(* IEC 61131-3 sources: Trae_CLoudTest/_archive/2026-04-25_全局规范修订V4.1.0/旧版程序文件, 5 files *)

(* ---- FB_单层输送机_V4.0.1.st ---- *)
//==============================================================================
// 边框缓存机 PLC程序 - 单层输送机纯逻辑功能块
// 版本: V4.0.1 (修正计时器使用方式 - 严格按三菱GX Works3标准)
// 项目: DJ-2026-005 边框缓存机
// 编制日期: 2026-04-23
// 更新日期: 2026-04-25 (修正计时器使用规范)
// 遵循规范: IEC 61131-3, 810_PLC编程规范_DEV-V1.0.0, 三菱GX Works3标准
//
// 说明:
//   纯逻辑功能块 - 单层输送机独立控制(不包含任何X/Y/M/D地址引用)
//   所有输入来自主控(已映射的逻辑变量), 所有输出给主控(由主控映射到Y地址)
//
// 功能:
//   1. 9步自动模式状态机控制
//   2. 手动模式点动控制(6个手动操作)
//   3. 初始化流程(气缸复位、状态清零)
//   4. 块内报警检测与处理(7种报警类型)
//   5. 完全自包含,无外部物理地址依赖,无ARRAY,纯单层设计
//
// 架构特点:
//   - 纯逻辑块: 不包含任何X/Y/M/D地址引用
//   - 数据解耦: 通过逻辑变量接口与主控交互
//   - 单层设计: 无ARRAY,所有信号均为单个BOOL/INT/REAL
//   - 故障安全: 内置超时保护和传感器冲突检测
//   - 下游联动: 支持上游允许放料信号和下游放料完成信号交互
//
// ⭐ 计时器使用规范 (V4.0.1 - 严格模仿三菱TIMER_100_FB_M_1):
//   参考原始程序:
//     TIMER_100_FB_M_1(MM[0] & NOT 异常暂停信号, 100, 0, TT1[0], MM[1]);
//     TIMER_100_FB_M_2(MM[2] & NOT 异常暂停信号, TT0[7], 0, TT1[1], MM[3]);
//
//   标准用法:
//     1. 程序开头统一调用TON实例(类似TIMER_100_FB_M_x调用)
//     2. 使用中间BOOL变量控制启动/停止(类似MM[x]:=1/0)
//     3. 使用中间BOOL变量判断到时(类似IF MM[y])
//     4. CASE状态机逻辑中只读写这些中间变量,不直接调用TON
//==============================================================================

FUNCTION_BLOCK FB_单层输送机_V4.0.1

VAR_INPUT
    (*==========================================================================
      一、系统控制信号 (来自主控/HMI M区) - 遵循801规范: i_前缀
      ==========================================================================*)
    i_bEnable            : BOOL;    // 总使能信号(主控系统就绪后置位)

    (*-------------------------------------------------------------------------
      模式选择 (互斥信号,来自HMI M区)
      -------------------------------------------------------------------------*)
    i_bAutoMode          : BOOL;    // 自动运行模式选择
    i_bManualMode        : BOOL;    // 手动调试模式选择

    (*-------------------------------------------------------------------------
      操作按钮 (来自HMI,边沿触发)
      -------------------------------------------------------------------------*)
    i_bStart             : BOOL;    // 自动循环启动按钮
    i_bStop              : BOOL;    // 自动循环停止按钮
    i_bReset             : BOOL;    // 故障复位/初始化按钮

    (*==========================================================================
      二、手动操作信号 (6个BOOL,来自HMI) - 遵循801规范: i_bLx_前缀(HMI辅助)
      ==========================================================================*)
    i_bLx_BlockDown      : BOOL;    // 手动-阻挡气缸下降
    i_bLx_BlockUp        : BOOL;    // 手动-阻挡气缸上升
    i_bLx_SeparatePush   : BOOL;    // 手动-分料气缸推出
    i_bLx_SeparateReset  : BOOL;    // 手动-分料气缸复位
    i_bLx_ConveyorFwd    : BOOL;    // 手动-输送带正转
    i_bLx_ConveyorRev    : BOOL;    // 手动-输送带反转

    (*==========================================================================
      三、工艺参数 (来自HMI设定或配方)
      ==========================================================================*)
    i_rConveyorSpeed     : REAL;    // 输送带速度设定(Hz或m/min,给变频器用)
    i_iSeparateTime      : INT;     // 分料动作保持时间(ms)
    i_iBlockWaitTime     : INT;     // 阻挡气缸动作等待时间(ms)

    (*==========================================================================
      四、传感器输入 (7个BOOL,全部来自主控映射)
      注: 放料完成感应器通过下游信号o_bFeedComplete反馈
      ==========================================================================*)
    (*--- 分料前感应器: 检测材料是否到达分料工位入口 ---*)
    i_bPreSeparateSensor : BOOL;

    (*--- 到位感应器1/2: 双传感器冗余检测材料到位 ---*)
    i_bPositionSensor1   : BOOL;
    i_bPositionSensor2   : BOOL;

    (*--- 阻挡气缸位置反馈 ---*)
    i_bBlockCylinderUp   : BOOL;    // 阻挡升起(释放)位置
    i_bBlockCylinderDown : BOOL;    // 阻挡下降(阻挡)位置

    (*--- 分料气缸位置反馈 ---*)
    i_bSeparateCylinderUp   : BOOL; // 分料收回位置
    i_bSeparateCylinderDown : BOOL; // 分料推出位置

    (*==========================================================================
      五、上下游联锁信号
      ==========================================================================*)
    i_bUpstreamAllowFeed : BOOL;    // 取放料机构已取走,允许继续放料
END_VAR

VAR_OUTPUT
    (*==========================================================================
      一、执行器请求输出 (5个BOOL,全部给主控,由主控映射到Y地址)
      ==========================================================================*)
    o_bBlockSolenoid     : BOOL;    // TRUE=下降(阻挡), FALSE=上升(释放)
    o_bSeparateSolenoid  : BOOL;    // TRUE=推出(分料), FALSE=复位
    o_bConveyorFwd       : BOOL;    // 输送带正向运转
    o_bConveyorSlow      : BOOL;    // 输送带慢速运转(精确定位用)
    o_bConveyorRev       : BOOL;    // 输送带反向运转(退料用)

    (*==========================================================================
      二、下游信号输出 (给取放料机构/打胶机)
      ==========================================================================*)
    o_bFeedComplete      : BOOL;    // 该层放料完成,可取料

    (*==========================================================================
      三、状态/HMI显示输出
      ==========================================================================*)
    o_bRunning           : BOOL;    // 正在自动运行
    o_bFault             : BOOL;    // 本站有故障(报警激活)
    o_iCurrentState      : INT;     // 当前状态码(0=空闲,1-8=步序,99=故障)

    (*==========================================================================
      四、报警输出 (给公共报警管理器)
      ==========================================================================*)
    o_iAlarmCode         : INT;     // 当前有效报警代码(0=无报警,1-7=报警类型)
                                    // 1=阻挡下降超时,2=上升超时,
                                    // 3=分料推出超时,4=复位超时,
                                    // 5=输送超时,6=传感器冲突,7=变频器故障
END_VAR

(*==============================================================================
 内部变量定义 - 遵循801规范: 不加前缀,直接 类型_描述
 ==============================================================================*)
VAR
    (*--------------------------------------------------------------------------
      一、状态机变量
      --------------------------------------------------------------------------*)
    iStep                : INT;     // 当前步序 (0-8)

    (*--- 运行标志 ---*)
    bRunning             : BOOL;    // 正在自动运行标志
    bFault               : BOOL;    // 故障标志

    (*--- 启动触发锁存 (防止重复触发) ---*)
    bStartTriggered       : BOOL;    // 启动信号锁存

    (*--------------------------------------------------------------------------
      二、⭐ 计时器相关变量 - 按三菱标准+801规范命名

      三菱标准接口:
        i_bTime  : BOOL  - 定时器启动输入 (Coil, 类似MM[x])
        q_bTq    : BOOL  - 定时器到时输出 (Status, 类似MM[y])
        i_bTrst  : BOOL  - 定时器复位信号
        i_pTimer : DINT - 定时器预设值 (Preset, 类似TT0[z])
        q_eTimer : DINT - 定时器当前值 (ValueOut, 类似TT1[w])

      801规范前缀:
        i_ = 输入变量 (VAR_INPUT风格,用于内部接口)
        q_ = 输出变量 (VAR_OUTPUT风格,用于内部接口)
      --------------------------------------------------------------------------*)

    (*--- TON计时器实例 (在VAR区声明,类似程序开头的TIMER_100_FB_M_x调用) ---*)
    tTimerAction         : TON;     // 动作等待定时器(阻挡/分料)
    tTimerConveyor       : TON;     // 输送超时定时器
    tTimerReset          : TON;     // 复位等待定时器
    tTimerPulse          : TON;     // 放料完成脉冲定时器(500ms)
    tTimerInit           : TON;     // 初始化总超时定时器

    (*--- 计时器接口变量 (严格按三菱标准命名) ---*)

    (* 启动输入: 写入TRUE=启动, 写入FALSE=停止 (类似 MM[x]:=1/0) *)
    i_bTime_Action       : BOOL;    // 动作定时器启动
    i_bTime_Conveyor     : BOOL;    // 输送定时器启动
    i_bTime_Reset        : BOOL;    // 复位定时器启动
    i_bTime_Pulse        : BOOL;    // 脉冲定时器启动
    i_bTime_Init         : BOOL;    // 初始化定时器启动

    (* 到时输出: 读取判断是否到时 (类似 IF MM[y]) *)
    q_bTq_Action         : BOOL;    // 动作定时器到时
    q_bTq_Conveyor       : BOOL;    // 输送定时器到时
    q_bTq_Reset          : BOOL;    // 复位定时器到时
    q_bTq_Pulse          : BOOL;    // 脉冲定时器到时
    q_bTq_Init           : BOOL;    // 初始化定时器到时

    (* 复位信号: 强制清零当前值 *)
    i_bTrst_Action       : BOOL;    // 动作定时器复位
    i_bTrst_Conveyor     : BOOL;    // 输送定时器复位

    (* 预设值: 可选,用于调试显示 (类似读取TT0[z]) *)
    i_pTimer_Action      : INT;     // 动作定时器预设值(ms)
    i_pTimer_Conveyor    : INT;     // 输送定时器预设值(ms)

    (* 当前值: 可选,用于调试显示 (类似读取TT1[w]) *)
    q_eTimer_Action      : INT;     // 动作定时器当前值(ms)
    q_eTimer_Conveyor    : INT;     // 输送定时器当前值(ms)

    (*--------------------------------------------------------------------------
      三、系统级内部变量
      --------------------------------------------------------------------------*)
    bInitComplete        : BOOL;    // 上电初始化完成标志
    bInitInProgress      : BOOL;    // 正在执行初始化

    (*--- 报警相关 ---*)
    iActiveAlarm         : INT;     // 当前活跃报警代码

    (*--- 传感器冲突检测 ---*)
    bBlockConflict       : BOOL;    // 阻挡上下位同时为TRUE
    bSeparateConflict    : BOOL;    // 分料上下位同时为TRUE

    (*--- 手动操作互锁 ---*)
    bManualAllow         : BOOL;    // 允许手动操作标志
END_VAR

(*==============================================================================
 常量定义 (状态机步序 + 报警码 + 定时参数)
 ==============================================================================*)
VAR CONSTANT
    (*--------------------------------------------------------------------------
      状态机步序常量 (9步: 0空闲 + 8工作步)
      --------------------------------------------------------------------------*)
    STP_IDLE             : INT := 0;   // 空闲待机
    STP_DETECT_MATERIAL  : INT := 1;   // 等待分料前感应器信号
    STP_BLOCK_DOWN       : INT := 2;   // 阻挡气缸下降到位
    STP_CONVEYOR_FWD     : INT := 3;   // 输送带正转运料
    STP_POSITION_CHECK   : INT := 4;   // 等待双传感器到位确认
    STP_BLOCK_UP         : INT := 5;   // 阻挡气缸上升释放
    STP_SEPARATE_ACTION  : INT := 6;   // 分料气缸推出分离
    STP_SLOW_FEED        : INT := 7;   // 慢速精确送出
    STP_FEED_COMPLETE    : INT := 8;   // 放料完成,等待取料

    (*--------------------------------------------------------------------------
      报警码常量 (1~7段,0=无报警)
      --------------------------------------------------------------------------*)
    ALM_BLOCK_DOWN_TIMEOUT   : INT := 1;
    ALM_BLOCK_UP_TIMEOUT    : INT := 2;
    ALM_SEPARATE_PUSH_TIMEOUT : INT := 3;
    ALM_SEPARATE_RESET_TIMEOUT : INT := 4;
    ALM_CONVEYOR_TIMEOUT    : INT := 5;
    ALM_SENSOR_CONFLICT     : INT := 6;
    ALM_INVERTER_FAULT      : INT := 7;

    (*--------------------------------------------------------------------------
      默认定时参数 (单位: ms,可通过输入参数覆盖)
      --------------------------------------------------------------------------*)
    T_DEF_BLOCK_ACTION_TIME     : INT := 800;    // 阻挡气缸动作时间
    T_DEF_SEPARATE_ACTION_TIME  : INT := 1000;   // 分料气缸动作时间
    T_DEF_CONVEYOR_TIMEOUT_TIME : INT := 5000;   // 输送带超时保护
    T_DEF_POSITION_STABLE_TIME  : INT := 500;    // 到位后稳定等待
    T_DEF_SLOW_FEED_TIME        : INT := 2000;   // 慢速送出时间
    T_DEF_RESET_WAIT_TIME       : INT := 500;    // 复位等待时间
    T_DEF_INIT_TIMEOUT          : INT := 10000;  // 初始化总超时(10s)
    T_DEF_FEED_PULSE_TIME       : INT := 500;    // 放料完成脉冲宽度(ms)
END_VAR

(*==============================================================================
 主程序开始 - 执行顺序说明 (严格模仿三菱原始程序结构):

   第一部分: 使能与初始化处理
   第二部分: 传感器冲突检测
   第三部分: 模式分发 (自动/手动)
   第四部分: 停止与复位处理
   第五部分: ⭐ TON统一实例化 (模仿TIMER_100_FB_M_x调用)
   第六部分: 状态机逻辑 (只操作bTimerXXX_Done接口,不直接调用TON)
   第七部分: 状态输出汇总
 ==============================================================================*)

//==============================================================================
// 第一部分: 使能与初始化处理
//==============================================================================

(*--- 使能失效时的安全处理 ---*)
IF NOT i_bEnable THEN
    (* 清零所有输出 *)
    o_bBlockSolenoid    := FALSE;
    o_bSeparateSolenoid := FALSE;
    o_bConveyorFwd      := FALSE;
    o_bConveyorSlow     := FALSE;
    o_bConveyorRev      := FALSE;
    o_bFeedComplete     := FALSE;

    (* 清零状态 *)
    iStep               := STP_IDLE;
    bRunning            := FALSE;
    bFault              := FALSE;
    bStartTriggered     := FALSE;
    iActiveAlarm        := 0;
    bInitComplete       := FALSE;
    bInitInProgress     := FALSE;

    (* 清零输出状态 *)
    o_bRunning          := FALSE;
    o_bFault            := FALSE;
    o_iCurrentState     := STP_IDLE;
    o_iAlarmCode        := 0;

    (* ⭐ 停止所有计时器 (清除启动标志,类似 MM[x]:=0) *)
    i_bTime_Action   := FALSE;
    i_bTime_Conveyor := FALSE;
    i_bTime_Reset    := FALSE;
    i_bTime_Pulse    := FALSE;
    i_bTime_Init     := FALSE;

    RETURN;  (* 退出功能块,不执行后续逻辑 *)
END_IF;

//==============================================================================
// 第二部分: 初始化流程 (上电或复位后首次使能时执行)
//==============================================================================

IF NOT bInitComplete THEN
    bInitInProgress := TRUE;

    (* ⭐ 启动初始化计时器 (设置启动标志,类似 MM[x]:=1) *)
    i_bTime_Init := TRUE;

    (* 执行初始化: 气缸回到安全位置 *)
    (* 阻挡电磁阀OFF -> 阻挡上升到上位 *)
    o_bBlockSolenoid    := FALSE;
    (* 分料电磁阀OFF -> 分料气缸复位到上位 *)
    o_bSeparateSolenoid := FALSE;
    (* 输送带全部停止 *)
    o_bConveyorFwd      := FALSE;
    o_bConveyorSlow     := FALSE;
    o_bConveyorRev      := FALSE;
    (* 步序归零 *)
    iStep               := STP_IDLE;
    bFault              := FALSE;
    iActiveAlarm        := 0;

    (* 检查初始化条件: 阻挡在上位 AND 分料在上位 OR 超时强制完成 *)
    IF (i_bBlockCylinderUp AND i_bSeparateCylinderUp) OR q_bTq_Init THEN
        (* 初始化完成 或 超时强制完成 *)
        bInitComplete   := TRUE;
        bInitInProgress := FALSE;
        (* ⭐ 停止初始化计时器 (清除启动标志,类似 MM[x]:=0) *)
        i_bTime_Init := FALSE;
    END_IF;

    (* 初始化期间不执行自动/手动逻辑 *)
    o_bRunning      := FALSE;
    o_iCurrentState := STP_IDLE;
    RETURN;
END_IF;

//==============================================================================
// 第三部分: 传感器冲突检测 (所有模式共用)
//==============================================================================

(* 阻挡气缸上下位同时为TRUE -> 传感器故障或接线错误 *)
bBlockConflict := i_bBlockCylinderUp AND i_bBlockCylinderDown;

(* 分料气缸上下位同时为TRUE -> 传感器故障或接线错误 *)
bSeparateConflict := i_bSeparateCylinderUp AND i_bSeparateCylinderDown;

(* 记录传感器冲突报警 *)
IF bBlockConflict OR bSeparateConflict THEN
    iActiveAlarm := ALM_SENSOR_CONFLICT;
    bFault      := TRUE;
ELSIF iActiveAlarm = ALM_SENSOR_CONFLICT THEN
    (* 冲突消失且当前只有此报警 -> 清除 *)
    iActiveAlarm := 0;
    bFault      := FALSE;
END_IF;

//==============================================================================
// 第四部分: 模式分发 (自动/手动)
//==============================================================================

IF i_bAutoMode THEN
    (*==========================================================================
      自动模式: 执行9步状态机
      =========================================================================*)
    CALL_AutoModeStateMachine();

ELSIF i_bManualMode THEN
    (*==========================================================================
      手动模式: 执行手动点动控制
      =========================================================================*)
    CALL_ManualModeControl();

ELSE
    (* 无效模式: 停止所有输出 *)
    o_bBlockSolenoid    := FALSE;
    o_bSeparateSolenoid := FALSE;
    o_bConveyorFwd      := FALSE;
    o_bConveyorSlow     := FALSE;
    o_bConveyorRev      := FALSE;
    o_bFeedComplete     := FALSE;

    (* 如果不在故障态,归零步序 *)
    IF NOT bFault THEN
        iStep := STP_IDLE;
    END_IF;
    bRunning := FALSE;

    (* ⭐ 无效模式下也停止所有计时器 *)
    i_bTime_Action   := FALSE;
    i_bTime_Conveyor := FALSE;
    i_bTime_Reset    := FALSE;
    i_bTime_Pulse    := FALSE;
END_IF;

//==============================================================================
// 第五部分: 停止与复位处理
//==============================================================================

(*--- 全局停止: 停止自动循环 ---*)
IF i_bStop THEN
    IF bRunning AND NOT bFault THEN
        iStep           := STP_IDLE;
        bRunning        := FALSE;
        bStartTriggered := FALSE;

        (* 停止该层输出 *)
        o_bBlockSolenoid    := FALSE;
        o_bSeparateSolenoid := FALSE;
        o_bConveyorFwd      := FALSE;
        o_bConveyorSlow     := FALSE;
        o_bConveyorRev      := FALSE;

        (* ⭐ 停止所有计时器 *)
        i_bTime_Action   := FALSE;
        i_bTime_Conveyor := FALSE;
        i_bTime_Reset    := FALSE;
        i_bTime_Pulse    := FALSE;
    END_IF;
END_IF;

(*--- 全局复位: 清除所有报警和故障 ---*)
IF i_bReset THEN
    IF bFault THEN
        (* 清除报警和故障标志 *)
        iActiveAlarm := 0;
        bFault      := FALSE;

        (* 归零步序 *)
        iStep           := STP_IDLE;
        bRunning        := FALSE;
        bStartTriggered := FALSE;

        (* 安全输出状态 *)
        o_bBlockSolenoid    := FALSE;
        o_bSeparateSolenoid := FALSE;
        o_bConveyorFwd      := FALSE;
        o_bConveyorSlow     := FALSE;
        o_bConveyorRev      := FALSE;
        o_bFeedComplete     := FALSE;

        (* ⭐ 停止所有计时器 *)
        i_bTime_Action   := FALSE;
        i_bTime_Conveyor := FALSE;
        i_bTime_Reset    := FALSE;
        i_bTime_Pulse    := FALSE;

        (* 要求重新初始化 *)
        bInitComplete := FALSE;
    END_IF;
END_IF;

//==============================================================================
// 第五部分: ⭐ TON统一实例化 (严格模仿三菱TIMER_100_FB_M_x模式)
//
// 原始程序格式:
//   TIMER_100_FB_M_1(MM[0] & NOT 异常暂停信号, 100, 0, TT1[0], MM[1]);
//   参数: s1(Coil)=执行条件, s2(Preset)=设定值, s3(ValueIn)=初始值,
//         d1(ValueOut)=当前值, d2(Status)=到时输出
//
// 本实现使用IEC标准TON,但保持相同的使用模式:
//   - 此处统一调用所有TON实例(类似程序开头的5行TIMER调用)
//   - 使用i_bTime_xxx控制IN(类似MM[x])
//   - 将.Q映射到q_bTq_xxx(类似MM[y])
//   - 将.ET映射到q_eTimer_xxx(类似TT1[w])
//==============================================================================

(*--- TON_1: 动作定时器 (阻挡/分料动作等待) ---*)
tTimerAction(
    IN  := i_bTime_Action,
    PT  := T#MS * (
            IF iStep = STP_BLOCK_DOWN AND i_iBlockWaitTime > 0
                THEN i_iBlockWaitTime
            ELSIF iStep = STP_SEPARATE_ACTION AND i_iSeparateTime > 0
                THEN i_iSeparateTime
            ELSIF iStep = STP_POSITION_CHECK
                THEN T_DEF_POSITION_STABLE_TIME
            ELSE
                T_DEF_BLOCK_ACTION_TIME
            END
        )
);

(*--- TON_2: 输送定时器 (输送超时保护) ---*)
tTimerConveyor(
    IN  := i_bTime_Conveyor,
    PT  := T#MS * (
            IF iStep = STP_SLOW_FEED
                THEN T_DEF_SLOW_FEED_TIME
            ELSE
                T_DEF_CONVEYOR_TIMEOUT_TIME
            END
        )
);

(*--- TON_3: 复位定时器 (暂未使用,预留) ---*)
tTimerReset(
    IN  := i_bTime_Reset,
    PT  := T#MS * T_DEF_RESET_WAIT_TIME
);

(*--- TON_4: 放料完成脉冲定时器 (500ms脉冲) ---*)
tTimerPulse(
    IN  := i_bTime_Pulse,
    PT  := T#MS * T_DEF_FEED_PULSE_TIME
);

(*--- TON_5: 初始化定时器 (10s总超时) ---*)
tTimerInit(
    IN  := i_bTime_Init,
    PT  := T#MS * T_DEF_INIT_TIMEOUT
);

(*--- 映射输出接口 (将TON的.Q/.ET映射到标准接口变量) ---*)

(* 到时输出: .Q -> q_bTq_xxx (类似 Status->MM[y]) *)
q_bTq_Action     := tTimerAction.Q;
q_bTq_Conveyor   := tTimerConveyor.Q;
q_bTq_Reset      := tTimerReset.Q;
q_bTq_Pulse      := tTimerPulse.Q;
q_bTq_Init       := tTimerInit.Q;

(* 当前值: .ET -> q_eTimer_xxx (类似 ValueOut->TT1[w]) *)
q_eTimer_Action   := UINT_TO_INT(TIME_TO_UINT(tTimerAction.ET)) / 10;   // 转换为ms
q_eTimer_Conveyor := UINT_TO_INT(TIME_TO_UINT(tTimerConveyor.ET)) / 10;

(* 预设值记录: PT -> i_pTimer_xxx (用于调试显示) *)
i_pTimer_Action   := UINT_TO_INT(TIME_TO_UINT(tTimerAction.PT)) / 10;
i_pTimer_Conveyor := UINT_TO_INT(TIME_TO_UINT(tTimerConveyor.PT)) / 10;

//==============================================================================
// 第六部分: 状态机逻辑 (只操作q_bTq_xxx接口,不直接调用TON)
// 类似原始程序的CASE Step_S OF ... END_CASE部分
//==============================================================================

(*--- 9步状态机主体 (仅使用q_bTq_xxx判断到时,类似IF MM[y]) ---*)
CASE iStep OF

(*======================================================================
 步骤0: 空闲待机
 条件: 启动触发 + 分料前有材料 + 上游允许放料
 ======================================================================*)
STP_IDLE:
    bRunning := FALSE;

    (* 安全输出状态 *)
    o_bBlockSolenoid    := FALSE;
    o_bSeparateSolenoid := FALSE;
    o_bConveyorFwd      := FALSE;
    o_bConveyorSlow     := FALSE;
    o_bConveyorRev      := FALSE;
    o_bFeedComplete     := FALSE;

    (* ⭐ 停止所有计时器 (设置启动标志=FALSE,类似 MM[x]:=0) *)
    i_bTime_Action   := FALSE;
    i_bTime_Conveyor := FALSE;
    i_bTime_Pulse    := FALSE;

    (* 启动条件:
       - 收到启动触发
       - 分料前有材料到位
       - 上游允许放料(取放料机构已取走上一次的材料)
    *)
    IF bStartTriggered AND i_bPreSeparateSensor AND i_bUpstreamAllowFeed THEN
        iStep    := STP_DETECT_MATERIAL;
        bRunning := TRUE;
        (* ⭐ 启动输送计时器 (设置启动标志=TRUE,类似 MM[x]:=1) *)
        i_bTime_Conveyor := TRUE;
    END_IF;

(*======================================================================
 步骤1: 检测材料到位 (双重确认)
 转出条件: 分料前感应器稳定信号
 超时条件: 材料未到达 -> ALM_CONVEYOR_TIMEOUT (检查q_bTq_Conveyor)
 ======================================================================*)
STP_DETECT_MATERIAL:
    (* 等待分料前感应器稳定信号 *)
    IF i_bPreSeparateSensor THEN
        (* 材料确认到位,进入阻挡下降 *)
        iStep := STP_BLOCK_DOWN;
        (* ⭐ 切换到动作计时器 (先停旧的,再启新的) *)
        i_bTime_Conveyor := FALSE;  // 停止输送计时器
        i_bTime_Action := TRUE;     // 启动动作计时器
    ELSIF q_bTq_Conveyor THEN  (* ✅ 读取到时标志,类似 IF MM[3] *)
        (* 超时: 材料未到达 *)
        iActiveAlarm := ALM_CONVEYOR_TIMEOUT;
        bFault       := TRUE;
        iStep        := STP_IDLE;
        bRunning     := FALSE;
        i_bTime_Conveyor := FALSE;  // 停止计时器
    END_IF;

(*======================================================================
 步骤2: 阻挡下降 (等待气缸下位信号或超时)
 动作: 保持o_bBlockSolenoid=TRUE
 转出条件: i_bBlockCylinderDown
 超时条件: ALM_BLOCK_DOWN_TIMEOUT (检查q_bTq_Action)
 ======================================================================*)
STP_BLOCK_DOWN:
    o_bBlockSolenoid := TRUE;  (* 保持下降 *)

    IF i_bBlockCylinderDown THEN
        (* 阻挡到位,转入输送 *)
        iStep := STP_CONVEYOR_FWD;
        o_bConveyorFwd := TRUE;
        (* ⭐ 切换到输送计时器 *)
        i_bTime_Action := FALSE;
        i_bTime_Conveyor := TRUE;
    ELSIF q_bTq_Action THEN  (* ✅ 读取到时标志,类似 IF MM[1] *)
        (* 超时: 阻挡未到位 *)
        iActiveAlarm := ALM_BLOCK_DOWN_TIMEOUT;
        bFault       := TRUE;
        o_bBlockSolenoid := FALSE;
        iStep        := STP_IDLE;
        bRunning     := FALSE;
        i_bTime_Action := FALSE;
    END_IF;

(*======================================================================
 步骤3: 输送正转 (将材料送到到位传感器位置)
 动作: 保持o_bConveyorFwd=TRUE
 转出条件: i_bPositionSensor1 AND i_bPositionSensor2 (双传感器冗余)
 超时条件: ALM_CONVEYOR_TIMEOUT (检查q_bTq_Conveyor)
 ======================================================================*)
STP_CONVEYOR_FWD:
    o_bConveyorFwd := TRUE;  (* 保持正转 *)

    (* 双传感器都到位 -> 输送成功 *)
    IF i_bPositionSensor1 AND i_bPositionSensor2 THEN
        iStep := STP_POSITION_CHECK;
        o_bConveyorFwd := FALSE;  (* 停止输送 *)
        (* ⭐ 切换到动作计时器(到位稳定等待) *)
        i_bTime_Conveyor := FALSE;
        i_bTime_Action := TRUE;
    ELSIF q_bTq_Conveyor THEN  (* ✅ 读取到时标志 *)
        (* 超时: 输送未到位 *)
        iActiveAlarm := ALM_CONVEYOR_TIMEOUT;
        bFault       := TRUE;
        o_bConveyorFwd := FALSE;
        iStep        := STP_IDLE;
        bRunning     := FALSE;
        i_bTime_Conveyor := FALSE;
    END_IF;

(*======================================================================
 步骤4: 到位检测 (短暂稳定等待后进入阻挡上升)
 动作: 保持阻挡,全部输出关闭,等待稳定
 转出条件: 定时器到期 (检查q_bTq_Action)
 ======================================================================*)
STP_POSITION_CHECK:
    (* 全部输出保持关闭,等待稳定,但保持阻挡 *)
    o_bBlockSolenoid := TRUE;  (* 保持阻挡 *)

    IF q_bTq_Action THEN  (* ✅ 读取到时标志 *)
        iStep := STP_BLOCK_UP;
        (* 开始阻挡上升(释放) *)
        o_bBlockSolenoid := FALSE;  (* OFF=上升 *)
        (* ⭐ 继续使用动作计时器(阻挡上升等待) - PT会自动根据iStep调整 *)
    END_IF;

(*======================================================================
 步骤5: 阻挡上升 (释放材料,准备分料)
 动作: 保持o_bBlockSolenoid=FALSE (上升状态)
 转出条件: i_bBlockCylinderUp
 超时条件: ALM_BLOCK_UP_TIMEOUT (检查q_bTq_Action)
 ======================================================================*)
STP_BLOCK_UP:
    o_bBlockSolenoid := FALSE;  (* 保持上升状态 *)

    IF i_bBlockCylinderUp THEN
        (* 阻挡已上升,进入分料 *)
        iStep := STP_SEPARATE_ACTION;
        o_bSeparateSolenoid := TRUE;  (* 推出分料 *)
        (* ⭐ 继续使用动作计时器(分料动作等待) *)
    ELSIF q_bTq_Action THEN  (* ✅ 读取到时标志 *)
        (* 超时: 阻挡未上升 *)
        iActiveAlarm := ALM_BLOCK_UP_TIMEOUT;
        bFault       := TRUE;
        iStep        := STP_IDLE;
        bRunning     := FALSE;
        i_bTime_Action := FALSE;
    END_IF;

(*======================================================================
 步骤6: 分料动作 (分料气缸推出,将材料分离)
 动作: 保持o_bSeparateSolenoid=TRUE
 转出条件: i_bSeparateCylinderDown
 超时条件: ALM_SEPARATE_PUSH_TIMEOUT (检查q_bTq_Action)
 ======================================================================*)
STP_SEPARATE_ACTION:
    o_bSeparateSolenoid := TRUE;  (* 保持推出 *)

    IF i_bSeparateCylinderDown THEN
        (* 分料到位,转入慢速送出 *)
        iStep := STP_SLOW_FEED;
        o_bSeparateSolenoid := FALSE;  (* 开始复位 *)
        o_bConveyorSlow := TRUE;  (* 慢速送出 *)
        (* ⭐ 切换到输送计时器(慢速送出等待) *)
        i_bTime_Action := FALSE;
        i_bTime_Conveyor := TRUE;
    ELSIF q_bTq_Action THEN  (* ✅ 读取到时标志 *)
        (* 超时: 分料未到位 *)
        iActiveAlarm := ALM_SEPARATE_PUSH_TIMEOUT;
        bFault       := TRUE;
        o_bSeparateSolenoid := FALSE;
        iStep        := STP_IDLE;
        bRunning     := FALSE;
        i_bTime_Action := FALSE;
    END_IF;

(*======================================================================
 步骤7: 慢速送出 (精确送出到取料位置)
 动作: o_bConveyorSlow=TRUE, o_bSeparateSolenoid=FALSE(持续复位)
 转出条件: 定时器到期 + 分料已复位验证 (检查q_bTq_Conveyor)
 超时/异常: ALM_SEPARATE_RESET_TIMEOUT
 ======================================================================*)
STP_SLOW_FEED:
    o_bConveyorSlow     := TRUE;   (* 保持慢速 *)
    o_bSeparateSolenoid := FALSE;  (* 分料持续复位 *)

    (* 检查慢速送出时间到 *)
    IF q_bTq_Conveyor THEN  (* ✅ 读取到时标志 *)

        (* 验证分料气缸是否已复位 *)
        IF NOT i_bSeparateCylinderDown OR i_bSeparateCylinderUp THEN
            (* 正常: 分料已复位或在下位信号消失 *)
            iStep := STP_FEED_COMPLETE;
            o_bConveyorSlow := FALSE;
            o_bFeedComplete := TRUE;  (* 通知下游可取料 *)
            (* ⭐ 切换到脉冲计时器 *)
            i_bTime_Conveyor := FALSE;
            i_bTime_Pulse := TRUE;
        ELSE
            (* 异常: 分料气缸卡在推出位置 *)
            iActiveAlarm := ALM_SEPARATE_RESET_TIMEOUT;
            bFault       := TRUE;
            o_bConveyorSlow := FALSE;
            iStep        := STP_IDLE;
            bRunning     := FALSE;
            i_bTime_Conveyor := FALSE;
        END_IF;
    END_IF;

(*======================================================================
 步骤8: 放料完成 (等待下游取料完成后回到空闲)
 动作: 保持o_bFeedComplete=TRUE (脉冲500ms或直到下游确认)
 转出条件: 启动触发被消耗(下一轮启动可重新开始)
 ======================================================================*)
STP_FEED_COMPLETE:
    (* 放料完成脉冲控制: 保持500ms后自动结束 *)
    IF q_bTq_Pulse THEN  (* ✅ 读取到时标志 *)
        iStep           := STP_IDLE;
        bRunning        := FALSE;
        o_bFeedComplete := FALSE;
        bStartTriggered := FALSE;  (* 消耗启动触发,准备接收下一次 *)
        i_bTime_Pulse := FALSE;  (* 停止脉冲计时器 *)
    ELSE
        o_bFeedComplete := TRUE;  (* 保持放料完成信号 *)
    END_IF;

ELSE
    (* 无效步序: 强制归零 *)
    iStep   := STP_IDLE;
    bRunning := FALSE;
    (* 停止所有计时器 *)
    i_bTime_Action   := FALSE;
    i_bTime_Conveyor := FALSE;
    i_bTime_Reset    := FALSE;
    i_bTime_Pulse    := FALSE;

END_CASE;

//==============================================================================
// 第七部分: 状态输出汇总
//==============================================================================

(*--- 运行中标志 ---*)
o_bRunning := bRunning;

(*--- 故障标志 ---*)
o_bFault := bFault;

(*--- 当前状态: 有故障则返回99,否则返回当前步序 ---*)
IF bFault THEN
    o_iCurrentState := 99;
ELSE
    o_iCurrentState := iStep;
END_IF;

(*--- 报警代码输出 ---*)
o_iAlarmCode := iActiveAlarm;

(*==============================================================================
 子程序: 自动模式状态机 (9步完整流程)
 注意: 实际的状态机逻辑已在第六部分的CASE语句中实现
 此子程序保留用于未来扩展或复杂逻辑封装
 ==============================================================================*)
METHOD CALL_AutoModeStateMachine : VOID
    (* 状态机主体已在主程序第六部分实现,此处无需重复代码 *)
    (* 如需封装,可将第六部分的CASE语句移至此处 *)
END_METHOD

(*==============================================================================
 子程序: 手动模式控制 (6个手动操作,带互锁和安全限制)
  ==============================================================================*)
METHOD CALL_ManualModeControl : VOID

    (* 故障层禁止手动操作 *)
    IF bFault THEN
        bManualAllow      := FALSE;
        o_bBlockSolenoid  := FALSE;
        o_bSeparateSolenoid := FALSE;
        o_bConveyorFwd    := FALSE;
        o_bConveyorSlow   := FALSE;
        o_bConveyorRev    := FALSE;
        iStep             := STP_IDLE;

        (* 停止所有计时器 *)
        i_bTime_Action   := FALSE;
        i_bTime_Conveyor := FALSE;
        i_bTime_Reset    := FALSE;
        i_bTime_Pulse    := FALSE;

        RETURN;
    END_IF;

    bManualAllow := TRUE;
    bRunning     := FALSE;
    iStep        := STP_IDLE;  (* 手动模式下步序显示为空闲 *)
    o_bFeedComplete := FALSE;

    (* 停止所有自动计时器 *)
    i_bTime_Action   := FALSE;
    i_bTime_Conveyor := FALSE;
    i_bTime_Pulse    := FALSE;

    (*======================================================================
     手动操作 - 阻挡气缸控制 (互锁: 下降/上升不能同时)
     ======================================================================*)
    IF i_bLx_BlockDown AND NOT i_bLx_BlockUp THEN
        (* 下降请求 *)
        o_bBlockSolenoid := TRUE;  (* 下降 *)
    ELSIF i_bLx_BlockUp AND NOT i_bLx_BlockDown THEN
        (* 上升请求 *)
        o_bBlockSolenoid := FALSE;  (* 上升 *)
    ELSE
        (* 无操作: 保持当前位置 *)
    END_IF;

    (*======================================================================
     手动操作 - 分料气缸控制 (互锁: 推出/复位不能同时)
     ======================================================================*)
    IF i_bLx_SeparatePush AND NOT i_bLx_SeparateReset THEN
        (* 推出请求 *)
        o_bSeparateSolenoid := TRUE;  (* 推出 *)
    ELSIF i_bLx_SeparateReset AND NOT i_bLx_SeparatePush THEN
        (* 复位请求 *)
        o_bSeparateSolenoid := FALSE;  (* 复位 *)
    ELSE
        (* 无操作 *)
    END_IF;

    (*======================================================================
     手动操作 - 输送带控制 (互锁: 正转/反转不能同时,慢速可叠加)
     ======================================================================*)
    IF i_bLx_ConveyorFwd AND NOT i_bLx_ConveyorRev THEN
        o_bConveyorFwd := TRUE;
        o_bConveyorRev := FALSE;
    ELSIF i_bLx_ConveyorRev AND NOT i_bLx_ConveyorFwd THEN
        o_bConveyorFwd := FALSE;
        o_bConveyorRev := TRUE;
    ELSE
        (* 正转/反转都没按: 停止输送 *)
        o_bConveyorFwd := FALSE;
        o_bConveyorRev := FALSE;
    END_IF;

    (* 慢速可作为独立控制或与正转叠加(根据实际工艺需求调整) *)
    (* 此处默认: 手动模式下慢速由外部单独控制或与正转联动 *)
    o_bConveyorSlow := FALSE;  (* 手动模式下默认不用慢速,可按需修改 *)

END_FUNCTION_BLOCK

//==============================================================================
// 程序结束
//==============================================================================

(* ---- FB_取放料机构_V4.0.0.st ---- *)
//==============================================================================
// 边框缓存机 PLC程序 - 取放料机构纯逻辑功能块
// 版本: V4.0.0
// 项目: DJ-2026-005 边框缓存机
// 编制日期: 2026-04-23
// 遵循规范: IEC 61131-3, 810_PLC编程规范_DEV-V1.0.0
// 说明: 纯逻辑功能块 - 取放料机构独立控制(不包含任何X/Y/M/D地址引用)
//       所有输入来自主控(已映射的逻辑变量), 所有输出给主控(由主控映射到Y地址)
//
// 核心工艺:
//   一次取两根边框(前后夹紧同时动作), 4层总共循环取2次
//   取料顺序: 第1次取L1+L2层, 第2次取L3+L4层
//   每次取料后移动到放料位置, 完成放料后通知下游(打胶机送料机构)
//
// 架构特点:
//   - 纯逻辑块: 不包含任何X/Y/M/D地址引用
//   - 数据解耦: 通过逻辑变量接口与主控交互
//   - 11步状态机: 完整的自动取放料循环控制
//   - 故障安全: 内置超时保护、伺服故障检测、传感器冲突检测
//   - 4层循环: 自动管理4层取放料进度, 循环2次完成全部取料
//==============================================================================

//==============================================================================
// 功能块: FB_取放料机构 - 取放料机构纯逻辑控制
// 功能:
//   1. 自动模式状态机(11步完整取放料循环)
//   2. 手动模式控制(14个手动操作信号)
//   3. 初始化流程(气缸复位、伺服使能、状态清零)
//   4. 块内报警检测与处理(8种报警类型, 101~199段)
//   5. 4层循环计数器(一次取两层, 循环2次取完4层)
//   6. 完全自包含, 无外部物理地址依赖
//==============================================================================
FUNCTION_BLOCK FB_1003_PickPlace_BufferFraming

VAR_INPUT
    (*==========================================================================
      一、系统控制信号 (来自主控/HMI M区)
      ==========================================================================*)
    i_b使能               : BOOL;    // 总使能信号(主控系统就绪后置位)

    (*-------------------------------------------------------------------------
      模式选择 (互斥信号,来自HMI M区)
      -------------------------------------------------------------------------*)
    i_b自动模式           : BOOL;    // 自动运行模式选择
    i_b手动模式           : BOOL;    // 手动调试模式选择

    (*-------------------------------------------------------------------------
      操作按钮 (来自HMI,边沿触发或电平有效)
      -------------------------------------------------------------------------*)
    i_b启动               : BOOL;    // 自动循环启动按钮(上升沿触发)
    i_b停止               : BOOL;    // 自动循环停止按钮(电平有效)
    i_b复位               : BOOL;    // 故障复位/初始化按钮(电平有效)

    (*==========================================================================
      二、手动操作信号 (14个BOOL,来自HMI)
      ==========================================================================*)
    (*--- 伺服点动控制 (4个) ---*)
    i_bZ轴点动上          : BOOL;    // 手动-Z轴向上点动
    i_bZ轴点动下          : BOOL;    // 手动-Z轴向下点动
    i_bX1轴点动前         : BOOL;    // 手动-X1轴向前点动(取料方向)
    i_bX1轴点动后         : BOOL;    // 手动-X1轴向后点动(放料方向)

    (*--- 气缸手动控制 (10个) ---*)
    (* 升降气缸: 双电磁阀控制 *)
    i_b升降上升           : BOOL;    // 手动-升降气缸上升
    i_b升降下降           : BOOL;    // 手动-升降气缸下降

    (* 前夹紧气缸: 双电磁阀控制(夹紧/松开) *)
    i_b前夹紧夹紧         : BOOL;    // 手动-前夹紧气缸夹紧
    i_b前夹紧松开         : BOOL;    // 手动-前夹紧气缸松开

    (* 后夹紧气缸: 双电磁阀控制(夹紧/松开) *)
    i_b后夹紧夹紧         : BOOL;    // 手动-后夹紧气缸夹紧
    i_b后夹紧松开         : BOOL;    // 手动-后夹紧气缸松开

    (* 前夹紧2气缸: 双电磁阀控制(夹紧/松开) - 第二组前夹爪 *)
    i_b前夹紧2夹紧        : BOOL;    // 手动-前夹紧2气缸夹紧
    i_b前夹紧2松开        : BOOL;    // 手动-前夹紧2气缸松开

    (* 后夹紧2气缸: 双电磁阀控制(夹紧/松开) - 第二组后夹爪 *)
    i_b后夹紧2夹紧        : BOOL;    // 手动-后夹紧2气缸夹紧
    i_b后夹紧2松开        : BOOL;    // 手动-后夹紧2气缸松开

    (*==========================================================================
      三、工艺参数 (来自HMI设定或配方)
      ==========================================================================*)
    (*--- 运动速度参数 (REAL) ---*)
    i_r取料速度           : REAL;    // 取料过程Z轴下降/上升速度(mm/s或%)
    i_r放料速度           : REAL;    // 放料过程Z轴下降/上升速度(mm/s或%)
    i_rZ轴速度            : REAL;    // Z轴通用运动速度设定(mm/s)
    i_rX1轴速度           : REAL;    // X1轴通用运动速度设定(mm/s)

    (*--- 动作时间参数 (INT, 单位: ms) ---*)
    i_i夹紧确认时间       : INT;     // 夹爪夹紧确认等待时间(ms)
    i_i升降动作时间       : INT;     // 升降气缸动作超时时间(ms)

    (*==========================================================================
      四、传感器输入 (26个BOOL,全部来自主控IO映射)
      注: 本功能块不直接读取X地址, 所有传感器由主控映射后传入
      ==========================================================================*)

    (*--- 气缸位置传感器 (10个磁性开关) ---*)
    (* 升降气缸: 动点=下降到位, 原点=上升到位 *)
    i_b升降_动点           : BOOL;    // 升降气缸下降到位(动点)
    i_b升降_原点           : BOOL;    // 升降气缸上升到位(原点)

    (* 前夹紧气缸: 动点=夹紧到位, 原点=松开到位 *)
    i_b前夹紧_动点         : BOOL;    // 前夹紧气缸夹紧到位(动点)
    i_b前夹紧_原点         : BOOL;    // 前夹紧气缸松开到位(原点)

    (* 后夹紧气缸: 动点=夹紧到位, 原点=松开到位 *)
    i_b后夹紧_动点         : BOOL;    // 后夹紧气缸夹紧到位(动点)
    i_b后夹紧_原点         : BOOL;    // 后夹紧气缸松开到位(原点)

    (* 前夹紧2气缸: 第二组前夹爪 *)
    i_b前夹紧2_动点        : BOOL;    // 前夹紧2气缸夹紧到位(动点)
    i_b前夹紧2_原点        : BOOL;    // 前夹紧2气缸松开到位(原点)

    (* 后夹紧2气缸: 第二组后夹爪 *)
    i_b后夹紧2_动点        : BOOL;    // 后夹紧2气缸夹紧到位(动点)
    i_b后夹紧2_原点        : BOOL;    // 后夹紧2气缸松开到位(原点)

    (*--- 产品检测传感器 (4个光电传感器) ---*)
    (* 一次取两根边框: 长边×2 + 短边×2 *)
    i_b长边1检测           : BOOL;    // 长边1存在检测(光电传感器)
    i_b长边2检测           : BOOL;    // 长边2存在检测(光电传感器)
    i_b短边1检测           : BOOL;    // 短边1存在检测(光电传感器)
    i_b短边2检测           : BOOL;    // 短边2存在检测(光电传感器)

    (*--- 伺服轴状态信号 (12个, 来自驱动器和限位开关) ---*)
    (* 原点信号 *)
    i_bZ轴_原点            : BOOL;    // Z轴伺服原点信号
    i_bX1轴_原点           : BOOL;    // X1轴伺服原点信号
    i_bX2轴_原点           : BOOL;    // X2轴伺服原点信号(预留)

    (* 伺服故障报警 *)
    i_bZ轴_伺服故障        : BOOL;    // Z轴伺服驱动器故障(ALM输出)
    i_bX1轴_伺服故障       : BOOL;    // X1轴伺服驱动器故障(ALM输出)
    i_bX2轴_伺服故障       : BOOL;    // X2轴伺服驱动器故障(预留)

    (* 限位开关信号 *)
    i_bZ轴_正向限位        : BOOL;    // Z轴正向限位(上限位)
    i_bZ轴_反向限位        : BOOL;    // Z轴反向限位(下限位)
    i_bX1轴_正向限位       : BOOL;    // X1轴正向限位(取料侧限位)
    i_bX1轴_反向限位       : BOOL;    // X1轴反向限位(放料侧限位)
    i_bX2轴_正向限位       : BOOL;    // X2轴正向限位(预留)
    i_bX2轴_反向限位       : BOOL;    // X2轴反向限位(预留)

    (*==========================================================================
      五、上游信号 (来自四层输送机的放料完成信号)
      ==========================================================================*)
    i_b输送机_L1_放料完成  : BOOL;    // 输送机第1层放料完成
    i_b输送机_L2_放料完成  : BOOL;    // 输送机第2层放料完成
    i_b输送机_L3_放料完成  : BOOL;    // 输送机第3层放料完成
    i_b输送机_L4_放料完成  : BOOL;    // 输送机第4层放料完成
END_VAR

VAR_OUTPUT
    (*==========================================================================
      一、执行器请求输出 (给主控, 由主控映射到Y地址)
      ==========================================================================*)

    (*--- 气缸控制输出 (6个BOOL) ---*)
    (* 升降气缸: 上升/下降双电磁阀 *)
    o_b升降_上升           : BOOL;    // 升降气缸上升电磁阀 -> 主控 -> Y地址
    o_b升降_下降           : BOOL;    // 升降气缸下降电磁阀 -> 主控 -> Y地址

    (* 前夹紧气缸: 夹紧/松开双电磁阀 *)
    o_b前夹紧_夹紧         : BOOL;    // 前夹紧气缸夹紧电磁阀 -> 主控 -> Y地址
    o_b前夹紧_松开         : BOOL;    // 前夹紧气缸松开电磁阀 -> 主控 -> Y地址

    (* 后夹紧气缸: 夹紧/松开双电磁阀 *)
    o_b后夹紧_夹紧         : BOOL;    // 后夹紧气缸夹紧电磁阀 -> 主控 -> Y地址
    o_b后夹紧_松开         : BOOL;    // 后夹紧气缸松开电磁阀 -> 主控 -> Y地址

    (* 前夹紧2气缸: 夹紧/松开双电磁阀(第二组前夹爪) *)
    o_b前夹紧2_夹紧        : BOOL;    // 前夹紧2气缸夹紧电磁阀 -> 主控 -> Y地址
    o_b前夹紧2_松开        : BOOL;    // 前夹紧2气缸松开电磁阀 -> 主控 -> Y地址

    (* 后夹紧2气缸: 夹紧/松开双电磁阀(第二组后夹爪) *)
    o_b后夹紧2_夹紧        : BOOL;    // 后夹紧2气缸夹紧电磁阀 -> 主控 -> Y地址
    o_b后夹紧2_松开        : BOOL;    // 后夹紧2气缸松开电磁阀 -> 主控 -> Y地址

    (*--- 伺服控制输出 (3个BOOL, 仅Z轴由本功能块直接控制) ---*)
    (* 注: X1轴/X2轴的运动指令通过内部标志传递给主控处理脉冲输出 *)
    o_bZ轴_脉冲输出        : BOOL;    // Z轴脉冲输出使能 -> 主控 -> Y0(PULSE)
    o_bZ轴_方向输出        : BOOL;    // Z轴方向控制 -> 主控 -> Y4(SIGN)
    o_bZ轴_伺服使能        : BOOL;    // Z轴伺服励磁(SON) -> 主控 -> Y10

    (*==========================================================================
      二、下游信号输出 (给打胶机送料机构)
      ==========================================================================*)
    o_b放料完成_给送料机构 : BOOL;    // 放料完成通知下游(打胶机可取料)

    (*==========================================================================
      三、状态/HMI显示输出
      ==========================================================================*)
    o_b运行中             : BOOL;    // 本站正在自动运行
    o_b故障               : BOOL;    // 本站有故障(任一报警激活)
    o_i当前状态           : INT;     // 当前状态机步序(0~10, 99=故障)
    o_rZ轴当前位置        : REAL;    // Z轴当前位置反馈(mm, 来自主控映射)
    o_rX1轴当前位置       : REAL;    // X1轴当前位置反馈(mm, 来自主控映射)
    o_rX2轴当前位置       : REAL;    // X2轴当前位置反馈(mm, 预留, 来自主控映射)
    o_i当前取料层数       : INT;     // 当前正在处理的层数(0=空闲, 1~4=层号)

    (*==========================================================================
      四、报警输出 (给公共报警管理器)
      ==========================================================================*)
    o_i本站报警代码       : INT;     // 本站当前有效报警代码(0=无报警, 101~199=报警类型)
END_VAR

(*==============================================================================
 内部变量定义
 ==============================================================================*)
VAR
    (*--------------------------------------------------------------------------
      一、状态机核心变量
      --------------------------------------------------------------------------*)
    s_i步序               : INT;     // 当前状态机步序(0~10)
    s_b运行中             : BOOL;    // 自动运行中标志
    s_b故障               : BOOL;    // 故障标志
    s_b启动触发           : BOOL;    // 启动信号锁存(防重复触发)

    (*--- 4层循环计数器 ---*)
    s_i已完成层数         : INT;     // 已完成的取放料层数(0~4)
    s_i当前取料层号       : INT;     // 当前正在取料的层号(1~4)
    s_i取料次数           : INT;     // 当前是第几次取料(1或2)

    (*--- 放料完成通知脉冲 ---*)
    s_b放料完成脉冲       : BOOL;    // 放料完成单周期脉冲
    s_t放料完成保持定时器 : TON;     // 放料完成信号保持定时器

    (*--------------------------------------------------------------------------
      二、定时器 (覆盖所有时序需求)
      --------------------------------------------------------------------------*)
    s_t动作定时器         : TON;     // 通用动作等待定时器(升降/夹紧/松开/移动)
    s_t产品检测稳定定时器 : TON;     // 产品检测稳定等待定时器
    s_t初始化定时器       : TON;     // 初始化总超时定时器

    (*--------------------------------------------------------------------------
      三、系统级内部变量
      --------------------------------------------------------------------------*)
    s_b初始化完成         : BOOL;    // 上电初始化完成标志
    s_b初始化中           : BOOL;    // 正在执行初始化
    s_b产品检测通过       : BOOL;    // 产品检测结果(4传感器全检测到)

    (*--- 报警相关 ---*)
    s_i活跃报警           : INT;     // 当前最高优先级报警代码

    (*--- 伺服运动请求标志 (给主控处理脉冲输出) ---*)
    s_bZ轴请求下降        : BOOL;    // Z轴下降运动请求
    s_bZ轴请求上升        : BOOL;    // Z轴上升运动请求
    s_bX1轴请求前移       : BOOL;    // X1轴向前移动请求(去取料位置)
    s_bX1轴请求后移       : BOOL;    // X1轴向后移动请求(去放料位置)
    s_bX1轴在取料位       : BOOL;    // X1轴是否在取料位置标志
    s_bX1轴在放料位       : BOOL;    // X1轴是否在放料位置标志

    (*--- 传感器冲突检测 ---*)
    s_b升降冲突           : BOOL;    // 升降上下位同时为TRUE
    s_b前夹紧冲突         : BOOL;    // 前夹紧夹紧/松开同时为TRUE
    s_b后夹紧冲突         : BOOL;    // 后夹紧夹紧/松开同时为TRUE
    s_b前夹紧2冲突        : BOOL;    // 前夹紧2夹紧/松开同时为TRUE
    s_b后夹紧2冲突        : BOOL;    // 后夹紧2夹紧/松开同时为TRUE

    (*--- 手动操作互锁 ---*)
    s_b手动允许           : BOOL;    // 允许手动操作标志
END_VAR

(*==============================================================================
 常量定义 (状态机步序 + 报警码 + 定时参数)
 ==============================================================================*)
VAR CONSTANT
    (*--------------------------------------------------------------------------
      状态机步序常量 (11步: 0空闲 + 10工作步)
      核心工艺: 一次取两根边框, 4层循环取2次
      --------------------------------------------------------------------------*)
    STP_空闲              : INT := 0;   // 空闲待机
    STP_等待放料完成      : INT := 1;   // 等待输送机放料完成信号
    STP_取料下降          : INT := 2;   // Z轴下降到取料高度
    STP_夹爪夹紧          : INT := 3;   // 前后夹紧同时夹紧(一次取两根)
    STP_产品检测          : INT := 4;   // 产品检测确认(长边+短边共4传感器)
    STP_取料上升          : INT := 5;   // Z轴上升到安全高度
    STP_移动到放料位置    : INT := 6;   // X1轴移动到放料位置(打胶机侧)
    STP_放料下降          : INT := 7;   // Z轴下降到放料高度
    STP_夹爪松开          : INT := 8;   // 前后夹紧同时松开
    STP_放料上升          : INT := 9;   // Z轴上升到安全高度
    STP_放料完成通知      : INT := 10;  // 发送放料完成信号给下游

    (*--------------------------------------------------------------------------
      报警码常量 (101~199段, 0=无报警)
      与四层输送机(1~7段)、其他设备错开, 便于公共报警管理器区分来源
      --------------------------------------------------------------------------*)
    ALM_Z轴伺服故障       : INT := 101;  // Z轴伺服驱动器故障
    ALM_X1轴伺服故障      : INT := 102;  // X1轴伺服驱动器故障
    ALM_升降下降超时      : INT := 103;  // 升降气缸下降未到位
    ALM_升降上升超时      : INT := 104;  // 升降气缸上升未到位
    ALM_夹紧超时          : INT := 105;  // 夹爪夹紧未到位
    ALM_松开超时          : INT := 106;  // 夹爪松开未到位
    ALM_产品检测失败      : INT := 107;  // 产品检测失败(缺长边或短边)
    ALM_移动超时          : INT := 108;  // X1轴移动超时

    (*--------------------------------------------------------------------------
      默认定时参数 (单位: ms, 可通过输入参数覆盖)
      --------------------------------------------------------------------------*)
    T_DEF_升降动作时间    : INT := 2000;    // 升降气缸动作时间(上下行程)
    T_DEF_夹紧确认时间    : INT := 800;     // 夹爪夹紧确认时间
    T_DEF_松开确认时间    : INT := 800;     // 夹爪松开确认时间
    T_DEF_产品检测稳定时间 : INT := 300;    // 产品检测稳定等待时间
    T_DEF_移动超时时间    : INT := 5000;    // X1轴移动超时保护
    T_DEF_放料完成保持时间 : INT := 500;    // 放料完成信号保持时间
    T_DEF_初始化超时      : INT := 10000;   // 初始化总超时(10s)

    (*--- 层数常量 ---*)
    LAYER_TOTAL           : INT := 4;       // 总层数
    PICK_TIMES            : INT := 2;       // 取料次数(每次取2层, 共2次取完4层)
END_VAR

(*==============================================================================
 主程序开始
 ==============================================================================*)

//==============================================================================
// 第一部分: 使能与初始化处理
//==============================================================================

(*--- 使能失效时的安全处理: 全部输出归零, 状态复位 ---*)
IF NOT i_b使能 THEN
    (* 清零所有气缸输出 *)
    o_b升降_上升           := FALSE;
    o_b升降_下降           := FALSE;
    o_b前夹紧_夹紧         := FALSE;
    o_b前夹紧_松开         := FALSE;
    o_b后夹紧_夹紧         := FALSE;
    o_b后夹紧_松开         := FALSE;
    o_b前夹紧2_夹紧        := FALSE;
    o_b前夹紧2_松开        := FALSE;
    o_b后夹紧2_夹紧        := FALSE;
    o_b后夹紧2_松开        := FALSE;

    (* 清零所有伺服输出 *)
    o_bZ轴_脉冲输出        := FALSE;
    o_bZ轴_方向输出        := FALSE;
    o_bZ轴_伺服使能        := FALSE;

    (* 清零下游信号 *)
    o_b放料完成_给送料机构 := FALSE;

    (* 清零所有状态 *)
    s_i步序               := STP_空闲;
    s_b运行中             := FALSE;
    s_b故障               := FALSE;
    s_b启动触发           := FALSE;
    s_i已完成层数         := 0;
    s_i当前取料层号       := 0;
    s_i取料次数           := 0;
    s_b放料完成脉冲       := FALSE;
    s_b产品检测通过       := FALSE;

    (* 清零运动请求 *)
    s_bZ轴请求下降        := FALSE;
    s_bZ轴请求上升        := FALSE;
    s_bX1轴请求前移       := FALSE;
    s_bX1轴请求后移       := FALSE;
    s_bX1轴在取料位       := FALSE;
    s_bX1轴在放料位       := FALSE;

    (* 清零报警 *)
    s_i活跃报警           := 0;
    o_i本站报警代码       := 0;
    o_b故障               := FALSE;
    s_b初始化完成         := FALSE;
    s_b初始化中           := FALSE;

    (* 清零状态输出 *)
    o_b运行中             := FALSE;
    o_i当前状态           := STP_空闲;
    o_i当前取料层数       := 0;

    (* 停止所有定时器 *)
    s_t动作定时器(IN := FALSE);
    s_t产品检测稳定定时器(IN := FALSE);
    s_t初始化定时器(IN := FALSE);
    s_t放料完成保持定时器(IN := FALSE);

    RETURN;  (* 退出功能块, 不执行后续逻辑 *)
END_IF;

//==============================================================================
// 第二部分: 初始化流程 (上电或复位后首次使能时执行)
//==============================================================================

IF NOT s_b初始化完成 THEN
    s_b初始化中 := TRUE;

    (* 初始化定时器: 防止初始化卡死 *)
    s_t初始化定时器(IN := TRUE, PT := T_DEF_初始化超时);

    (* 初始化动作:
       1. 所有气缸回到安全位置(上升/松开状态)
       2. 伺服使能(准备回原点或保持当前位置)
       3. 状态清零
    *)

    (* 气缸安全位置: 升降上升, 所有夹紧松开 *)
    o_b升降_上升           := TRUE;   (* 上升 *)
    o_b升降_下降           := FALSE;
    o_b前夹紧_夹紧         := FALSE;
    o_b前夹紧_松开         := TRUE;   (* 松开 *)
    o_b后夹紧_夹紧         := FALSE;
    o_b后夹紧_松开         := TRUE;   (* 松开 *)
    o_b前夹紧2_夹紧        := FALSE;
    o_b前夹紧2_松开        := TRUE;   (* 松开 *)
    o_b后夹紧2_夹紧        := FALSE;
    o_b后夹紧2_松开        := TRUE;   (* 松开 *)

    (* 伺服使能: 使能Z轴伺服(实际回原点由主控统一协调) *)
    o_bZ轴_伺服使能        := TRUE;
    o_bZ轴_脉冲输出        := FALSE;
    o_bZ轴_方向输出        := FALSE;

    (* 下游信号清零 *)
    o_b放料完成_给送料机构 := FALSE;

    (* 步序归零 *)
    s_i步序               := STP_空闲;
    s_b故障               := FALSE;
    s_i活跃报警           := 0;

    (* 检查初始化条件:
       升降在原点(上位) AND 所有夹紧在原点(松开位)
       或 超时强制完成(允许在有报警情况下继续, 报警单独处理)
    *)
    IF (i_b升降_原点 AND
        i_b前夹紧_原点 AND i_b后夹紧_原点 AND
        i_b前夹紧2_原点 AND i_b后夹紧2_原点)
       OR s_t初始化定时器.Q THEN
        (* 初始化完成 或 超时强制完成 *)
        s_b初始化完成 := TRUE;
        s_b初始化中 := FALSE;
        s_t初始化定时器(IN := FALSE);

        (* 初始化完成后关闭气缸输出(进入空闲态的安全状态) *)
        o_b升降_上升       := FALSE;
        o_b前夹紧_松开     := FALSE;
        o_b后夹紧_松开     := FALSE;
        o_b前夹紧2_松开    := FALSE;
        o_b后夹紧2_松开    := FALSE;
    END_IF;

    (* 初始化期间不执行自动/手动逻辑 *)
    o_b运行中 := FALSE;
    o_i当前状态 := STP_空闲;
    o_i当前取料层数 := 0;
    RETURN;
END_IF;

//==============================================================================
// 第三部分: 伺服故障检测 (所有模式共用, 最高优先级)
//==============================================================================

(*--- Z轴伺服故障检测 ---*)
IF i_bZ轴_伺服故障 THEN
    IF s_i活跃报警 <> ALM_Z轴伺服故障 THEN
        s_i活跃报警 := ALM_Z轴伺服故障;
        s_b故障 := TRUE;
    END_IF;
    (* 伺服故障时立即停止Z轴输出 *)
    o_bZ轴_脉冲输出 := FALSE;
ELSIF s_i活跃报警 = ALM_Z轴伺服故障 THEN
    (* 故障消失且当前只有此报警 -> 清除 *)
    s_i活跃报警 := 0;
    s_b故障 := FALSE;
END_IF;

(*--- X1轴伺服故障检测 ---*)
IF i_bX1轴_伺服故障 THEN
    IF s_i活跃报警 <> ALM_X1轴伺服故障 THEN
        s_i活跃报警 := ALM_X1轴伺服故障;
        s_b故障 := TRUE;
    END_IF;
ELSIF s_i活跃报警 = ALM_X1轴伺服故障 THEN
    s_i活跃报警 := 0;
    s_b故障 := FALSE;
END_IF;

//==============================================================================
// 第四部分: 传感器冲突检测 (所有模式共用)
//==============================================================================

(*--- 升降气缸传感器冲突: 上下位同时为TRUE ---*)
s_b升降冲突 := i_b升降_动点 AND i_b升降_原点;
IF s_b升降冲突 THEN
    IF s_i活跃报警 = 0 OR s_i活跃报警 > ALM_产品检测失败 THEN
        (* 传感器冲突优先级低于动作超时, 但仍需记录 *)
        (* 此处暂不设独立报警码, 可扩展为109号 *)
    END_IF;
END_IF;

(*--- 各夹紧气缸传感器冲突检测 ---*)
s_b前夹紧冲突 := i_b前夹紧_动点 AND i_b前夹紧_原点;
s_b后夹紧冲突 := i_b后夹紧_动点 AND i_b后夹紧_原点;
s_b前夹紧2冲突 := i_b前夹紧2_动点 AND i_b前夹紧2_原点;
s_b后夹紧2冲突 := i_b后夹紧2_动点 AND i_b后夹紧2_原点;

//==============================================================================
// 第五部分: 模式分发 (自动/手动)
//==============================================================================

IF i_b自动模式 THEN
    (*==========================================================================
      自动模式: 执行11步取放料状态机
      =========================================================================*)
    CALL_自动模式状态机();

ELSIF i_b手动模式 THEN
    (*==========================================================================
      手动模式: 执行手动点动控制
      =========================================================================*)
    CALL_手动模式控制();

ELSE
    (* 无效模式: 停止所有输出, 进入安全状态 *)
    o_b升降_上升           := FALSE;
    o_b升降_下降           := FALSE;
    o_b前夹紧_夹紧         := FALSE;
    o_b前夹紧_松开         := FALSE;
    o_b后夹紧_夹紧         := FALSE;
    o_b后夹紧_松开         := FALSE;
    o_b前夹紧2_夹紧        := FALSE;
    o_b前夹紧2_松开        := FALSE;
    o_b后夹紧2_夹紧        := FALSE;
    o_b后夹紧2_松开        := FALSE;
    o_bZ轴_脉冲输出        := FALSE;
    o_bZ轴_方向输出        := FALSE;
    o_b放料完成_给送料机构 := FALSE;
    s_bZ轴请求下降        := FALSE;
    s_bZ轴请求上升        := FALSE;
    s_bX1轴请求前移       := FALSE;
    s_bX1轴请求后移       := FALSE;

    (* 如果不在故障态, 归零步序 *)
    IF NOT s_b故障 THEN
        s_i步序 := STP_空闲;
        s_b运行中 := FALSE;
    END_IF;
END_IF;

//==============================================================================
// 第六部分: 停止与复位处理
//==============================================================================

(*--- 全局停止: 停止自动循环, 保持当前位置 ---*)
IF i_b停止 THEN
    IF s_b运行中 AND NOT s_b故障 THEN
        (* 停止并复位到空闲 *)
        s_i步序 := STP_空闲;
        s_b运行中 := FALSE;
        s_b启动触发 := FALSE;

        (* 停止所有输出 *)
        o_b升降_上升           := FALSE;
        o_b升降_下降           := FALSE;
        o_b前夹紧_夹紧         := FALSE;
        o_b前夹紧_松开         := FALSE;
        o_b后夹紧_夹紧         := FALSE;
        o_b后夹紧_松开         := FALSE;
        o_b前夹紧2_夹紧        := FALSE;
        o_b前夹紧2_松开        := FALSE;
        o_b后夹紧2_夹紧        := FALSE;
        o_b后夹紧2_松开        := FALSE;
        o_b前夹紧2_夹紧        := FALSE;
        o_b前夹紧2_松开        := FALSE;
        o_b后夹紧2_夹紧        := FALSE;
        o_b后夹紧2_松开        := FALSE;
        o_bZ轴_脉冲输出        := FALSE;
        o_bZ轴_方向输出        := FALSE;
        o_b放料完成_给送料机构 := FALSE;

        (* 停止运动请求 *)
        s_bZ轴请求下降        := FALSE;
        s_bZ轴请求上升        := FALSE;
        s_bX1轴请求前移       := FALSE;
        s_bX1轴请求后移       := FALSE;

        (* 停止定时器 *)
        s_t动作定时器(IN := FALSE);
        s_t产品检测稳定定时器(IN := FALSE);
        s_t放料完成保持定时器(IN := FALSE);
    END_IF;
END_IF;

(*--- 全局复位: 清除所有报警和故障, 重新初始化 ---*)
IF i_b复位 THEN
    IF s_b故障 THEN
        (* 清除报警和故障标志 *)
        s_i活跃报警 := 0;
        s_b故障 := FALSE;
        o_i本站报警代码 := 0;

        (* 归零步序和计数器 *)
        s_i步序 := STP_空闲;
        s_b运行中 := FALSE;
        s_b启动触发 := FALSE;
        s_i已完成层数 := 0;
        s_i当前取料层号 := 0;
        s_i取料次数 := 0;
        s_b放料完成脉冲 := FALSE;
        s_b产品检测通过 := FALSE;

        (* 安全输出状态: 全部归零 *)
        o_b升降_上升           := FALSE;
        o_b升降_下降           := FALSE;
        o_b前夹紧_夹紧         := FALSE;
        o_b前夹紧_松开         := FALSE;
        o_b后夹紧_夹紧         := FALSE;
        o_b后夹紧_松开         := FALSE;
        o_b前夹紧2_夹紧        := FALSE;
        o_b前夹紧2_松开        := FALSE;
        o_b后夹紧2_夹紧        := FALSE;
        o_b后夹紧2_松开        := FALSE;
        o_b前夹紧2_夹紧        := FALSE;
        o_b前夹紧2_松开        := FALSE;
        o_b后夹紧2_夹紧        := FALSE;
        o_b后夹紧2_松开        := FALSE;
        o_bZ轴_脉冲输出        := FALSE;
        o_bZ轴_方向输出        := FALSE;
        o_b放料完成_给送料机构 := FALSE;

        (* 停止运动请求 *)
        s_bZ轴请求下降        := FALSE;
        s_bZ轴请求上升        := FALSE;
        s_bX1轴请求前移       := FALSE;
        s_bX1轴请求后移       := FALSE;
        s_bX1轴在取料位       := FALSE;
        s_bX1轴在放料位       := FALSE;

        (* 停止定时器 *)
        s_t动作定时器(IN := FALSE);
        s_t产品检测稳定定时器(IN := FALSE);
        s_t放料完成保持定时器(IN := FALSE);

        (* 要求重新初始化 *)
        s_b初始化完成 := FALSE;
    END_IF;
END_IF;

//==============================================================================
// 第七部分: 状态输出汇总
//==============================================================================

(*--- 运行中标志 ---*)
o_b运行中 := s_b运行中;

(*--- 故障标志 ---*)
o_b故障 := s_b故障;

(*--- 当前状态码 ---*)
IF s_b故障 THEN
    o_i当前状态 := 99;  (* 故障状态显示99 *)
ELSE
    o_i当前状态 := s_i步序;
END_IF;

(*--- 当前取料层数 ---*)
IF s_b运行中 THEN
    o_i当前取料层数 := s_i当前取料层号;
ELSIF s_i已完成层数 >= LAYER_TOTAL THEN
    o_i当前取料层数 := 0;  (* 全部完成, 空闲 *)
ELSE
    o_i当前取料层数 := 0;  (* 空闲状态 *)
END_IF;

(*--- 本站报警代码 ---*)
o_i本站报警代码 := s_i活跃报警;

(*==============================================================================
 子程序: 自动模式状态机 (11步完整取放料循环)
   核心工艺: 一次取两根边框, 4层循环取2次
   取料顺序: 第1次取L1+L2(相邻两层), 第2次取L3+L4(相邻两层)
  ==============================================================================*)
METHOD CALL_自动模式状态机 : VOID

    (*--- 故障时不执行状态机 ---*)
    IF s_b故障 THEN
        s_b运行中 := FALSE;
        (* 故障安全输出: 全部停止 *)
        o_b升降_上升           := FALSE;
        o_b升降_下降           := FALSE;
        o_b前夹紧_夹紧         := FALSE;
        o_b前夹紧_松开         := FALSE;
        o_b后夹紧_夹紧         := FALSE;
        o_b后夹紧_松开         := FALSE;
        o_b前夹紧2_夹紧        := FALSE;
        o_b前夹紧2_松开        := FALSE;
        o_b后夹紧2_夹紧        := FALSE;
        o_b后夹紧2_松开        := FALSE;
        o_bZ轴_脉冲输出        := FALSE;
        o_bZ轴_方向输出        := FALSE;
        o_b放料完成_给送料机构 := FALSE;
        s_bZ轴请求下降        := FALSE;
        s_bZ轴请求上升        := FALSE;
        s_bX1轴请求前移       := FALSE;
        s_bX1轴请求后移       := FALSE;
        s_t动作定时器(IN := FALSE);
        s_t产品检测稳定定时器(IN := FALSE);
        RETURN;
    END_IF;

    (*--- 启动触发检测 (上升沿) ---*)
    IF i_b启动 AND NOT s_b启动触发 THEN
        s_b启动触发 := TRUE;
        (* 重置循环计数器 *)
        IF s_i已完成层数 >= LAYER_TOTAL THEN
            s_i已完成层数 := 0;
        END_IF;
        (* 计算当前取料次数和层号 *)
        s_i取料次数 := (s_i已完成层数 / 2) + 1;
        IF s_i取料次数 > PICK_TIMES THEN
            s_i取料次数 := 1;
            s_i已完成层数 := 0;
        END_IF;
    END_IF;

    (*--- 单例状态机 (全局唯一, 因为只有一个取放料机构) ---*)
    CASE s_i步序 OF

    (*======================================================================
     步骤0: 空闲待机
     等待启动触发, 收到启动后进入等待放料完成
     ======================================================================*)
    STP_空闲:
        s_b运行中 := FALSE;
        (* 安全输出状态: 全部归零 *)
        o_b升降_上升           := FALSE;
        o_b升降_下降           := FALSE;
        o_b前夹紧_夹紧         := FALSE;
        o_b前夹紧_松开         := FALSE;
        o_b后夹紧_夹紧         := FALSE;
        o_b后夹紧_松开         := FALSE;
        o_bZ轴_脉冲输出        := FALSE;
        o_bZ轴_方向输出        := FALSE;
        o_b放料完成_给送料机构 := FALSE;
        s_bZ轴请求下降        := FALSE;
        s_bZ轴请求上升        := FALSE;
        s_bX1轴请求前移       := FALSE;
        s_bX1轴请求后移       := FALSE;
        s_i当前取料层号       := 0;

        (* 启动条件: 收到启动触发 *)
        IF s_b启动触发 THEN
            s_i步序 := STP_等待放料完成;
            s_b运行中 := TRUE;
            (* 计算本次要取的层号 *)
            IF s_i已完成层数 < 2 THEN
                (* 第1次取料: 取L1+L2层 *)
                s_i当前取料层号 := 1;  (* 表示正在取第1-2层 *)
            ELSE
                (* 第2次取料: 取L3+L4层 *)
                s_i当前取料层号 := 3;  (* 表示正在取第3-4层 *)
            END_IF;
        END_IF;

    (*======================================================================
     步骤1: 等待输送机放料完成
     根据当前取料次数判断需要等待哪些层的放料完成信号
     第1次取料(L1+L2): 等待L1和L2都放料完成
     第2次取料(L3+L4): 等待L3和L4都放料完成
     ======================================================================*)
    STP_等待放料完成:
        (* 等待对应层的放料完成信号 *)
        IF s_i已完成层数 < 2 THEN
            (* 第1次: 等待L1和L2放料完成 *)
            IF i_b输送机_L1_放料完成 AND i_b输送机_L2_放料完成 THEN
                (* 两层都已放料完成, 可以开始取料 *)
                s_i步序 := STP_取料下降;
                (* 启动升降下降定时器 *)
                s_t动作定时器(IN := TRUE,
                    PT := UINT_TO_INT(TIME_TO_UINT(T#MS * i_i升降动作时间)));
                IF i_i升降动作时间 = 0 THEN
                    s_t动作定时器(PT := T_DEF_升降动作时间);
                END_IF;
                (* 请求Z轴下降 *)
                s_bZ轴请求下降 := TRUE;
                s_bZ轴请求上升 := FALSE;
                o_bZ轴_脉冲输出 := TRUE;
                o_bZ轴_方向输出 := TRUE;  (* 方向: 下降 *)
            END_IF;
        ELSE
            (* 第2次: 等待L3和L4放料完成 *)
            IF i_b输送机_L3_放料完成 AND i_b输送机_L4_放料完成 THEN
                s_i步序 := STP_取料下降;
                s_t动作定时器(IN := TRUE,
                    PT := UINT_TO_INT(TIME_TO_UINT(T#MS * i_i升降动作时间)));
                IF i_i升降动作时间 = 0 THEN
                    s_t动作定时器(PT := T_DEF_升降动作时间);
                END_IF;
                s_bZ轴请求下降 := TRUE;
                s_bZ轴请求上升 := FALSE;
                o_bZ轴_脉冲输出 := TRUE;
                o_bZ轴_方向输出 := TRUE;  (* 方向: 下降 *)
            END_IF;
        END_IF;

    (*======================================================================
     步骤2: 取料下降 (Z轴下降到取料高度)
     等待升降气缸动点(下位)信号或超时
     ======================================================================*)
    STP_取料下降:
        (* 保持Z轴下降输出 *)
        o_bZ轴_脉冲输出 := TRUE;
        o_bZ轴_方向输出 := TRUE;  (* 下降方向 *)
        o_b升降_下降 := TRUE;       (* 升降气缸下降辅助 *)
        o_b升降_上升 := FALSE;

        IF i_b升降_动点 THEN
            (* 升降下降到位, 转入夹紧步骤 *)
            s_t动作定时器(IN := FALSE);
            s_bZ轴请求下降 := FALSE;
            o_bZ轴_脉冲输出 := FALSE;
            o_b升降_下降 := FALSE;
            s_i步序 := STP_夹爪夹紧;
            (* 启动夹紧确认定时器 *)
            s_t动作定时器(IN := TRUE,
                PT := UINT_TO_INT(TIME_TO_UINT(T#MS * i_i夹紧确认时间)));
            IF i_i夹紧确认时间 = 0 THEN
                s_t动作定时器(PT := T_DEF_夹紧确认时间);
            END_IF;
            (* 同时夹紧前后夹爪(一次取两根) *)
            o_b前夹紧_夹紧 := TRUE;
            o_b后夹紧_夹紧 := TRUE;
        ELSIF s_t动作定时器.Q THEN
            (* 超时: 升降下降未到位 *)
            s_t动作定时器(IN := FALSE);
            s_i活跃报警 := ALM_升降下降超时;
            s_b故障 := TRUE;
            s_bZ轴请求下降 := FALSE;
            o_bZ轴_脉冲输出 := FALSE;
            o_b升降_下降 := FALSE;
            s_i步序 := STP_空闲;
            s_b运行中 := FALSE;
            s_b启动触发 := FALSE;
        END_IF;

    (*======================================================================
     步骤3: 夹爪夹紧 (前后夹紧同时动作, 一次取两根边框)
     等待夹紧确认时间到或传感器确认
     ======================================================================*)
    STP_夹爪夹紧:
        (* 保持夹紧输出: 前后夹紧同时夹紧 *)
        o_b前夹紧_夹紧 := TRUE;
        o_b后夹紧_夹紧 := TRUE;
        o_b前夹紧_松开 := FALSE;
        o_b后夹紧_松开 := FALSE;

        (* 夹紧到位判断: 时间到 OR 传感器确认(动点ON) *)
        IF s_t动作定时器.Q OR
           (i_b前夹紧_动点 AND i_b后夹紧_动点) THEN
            s_t动作定时器(IN := FALSE);
            s_i步序 := STP_产品检测;
            (* 启动产品检测稳定定时器 *)
            s_t产品检测稳定定时器(IN := TRUE,
                PT := T_DEF_产品检测稳定时间);
        ELSIF s_t动作定时器.Q AND
              NOT (i_b前夹紧_动点 AND i_b后夹紧_动点) THEN
            (* 超时且传感器未确认 -> 夹紧超时报警 *)
            (* 注意: 此处用第二个定时器Q判断, 实际上面已先判断Q *)
        END_IF;

        (* 夹紧超时检测: 如果定时器到但传感器没确认 *)
        IF s_t动作定时器.Q AND
           NOT (i_b前夹紧_动点 AND i_b后夹紧_动点) THEN
            s_t动作定时器(IN := FALSE);
            s_i活跃报警 := ALM_夹紧超时;
            s_b故障 := TRUE;
            o_b前夹紧_夹紧 := FALSE;
            o_b后夹紧_夹紧 := FALSE;
            s_i步序 := STP_空闲;
            s_b运行中 := FALSE;
            s_b启动触发 := FALSE;
        END_IF;

    (*======================================================================
     步骤4: 产品检测 (确认长边+短边共4个传感器都有信号)
     一次取两根边框: 需要2个长边+2个短边全部检测到
     ======================================================================*)
    STP_产品检测:
        (* 保持夹紧状态, 等待产品检测稳定 *)
        o_b前夹紧_夹紧 := TRUE;
        o_b后夹紧_夹紧 := TRUE;

        IF s_t产品检测稳定定时器.Q THEN
            s_t产品检测稳定定时器(IN := FALSE);

            (* 产品检测判断: 4个传感器全为TRUE *)
            s_b产品检测通过 :=
                i_b长边1检测 AND i_b长边2检测 AND
                i_b短边1检测 AND i_b短边2检测;

            IF s_b产品检测通过 THEN
                (* 产品检测通过, 转入取料上升 *)
                s_i步序 := STP_取料上升;
                (* 启动上升定时器 *)
                s_t动作定时器(IN := TRUE,
                    PT := UINT_TO_INT(TIME_TO_UINT(T#MS * i_i升降动作时间)));
                IF i_i升降动作时间 = 0 THEN
                    s_t动作定时器(PT := T_DEF_升降动作时间);
                END_IF;
                (* 请求Z轴上升 *)
                s_bZ轴请求上升 := TRUE;
                o_bZ轴_脉冲输出 := TRUE;
                o_bZ轴_方向输出 := FALSE;  (* 方向: 上升 *)
                o_b升降_上升 := TRUE;
                o_b前夹紧_夹紧 := FALSE;  (* 保持夹紧但关闭输出, 由机械自锁保持 *)
                o_b后夹紧_夹紧 := FALSE;
            ELSE
                (* 产品检测失败: 缺少长边或短边 *)
                s_i活跃报警 := ALM_产品检测失败;
                s_b故障 := TRUE;
                o_b前夹紧_夹紧 := FALSE;
                o_b后夹紧_夹紧 := FALSE;
                s_i步序 := STP_空闲;
                s_b运行中 := FALSE;
                s_b启动触发 := FALSE;
            END_IF;
        END_IF;

    (*======================================================================
     步骤5: 取料上升 (Z轴上升到安全高度)
     等待升降原点(上位)信号或超时
     ======================================================================*)
    STP_取料上升:
        (* 保持Z轴上升输出 *)
        o_bZ轴_脉冲输出 := TRUE;
        o_bZ轴_方向输出 := FALSE;  (* 上升方向 *)
        o_b升降_上升 := TRUE;
        o_b升降_下降 := FALSE;

        IF i_b升降_原点 THEN
            (* 上升到位, 转入移动到放料位置 *)
            s_t动作定时器(IN := FALSE);
            s_bZ轴请求上升 := FALSE;
            o_bZ轴_脉冲输出 := FALSE;
            o_b升降_上升 := FALSE;
            s_i步序 := STP_移动到放料位置;
            (* 启动移动超时定时器 *)
            s_t动作定时器(IN := TRUE, PT := T_DEF_移动超时时间);
            (* 请求X1轴向后移动(去放料位置) *)
            s_bX1轴请求前移 := FALSE;
            s_bX1轴请求后移 := TRUE;
            s_bX1轴在取料位 := FALSE;
        ELSIF s_t动作定时器.Q THEN
            (* 超时: 上升未到位 *)
            s_t动作定时器(IN := FALSE);
            s_i活跃报警 := ALM_升降上升超时;
            s_b故障 := TRUE;
            s_bZ轴请求上升 := FALSE;
            o_bZ轴_脉冲输出 := FALSE;
            o_b升降_上升 := FALSE;
            s_i步序 := STP_空闲;
            s_b运行中 := FALSE;
            s_b启动触发 := FALSE;
        END_IF;

    (*======================================================================
     步骤6: 移动到放料位置 (X1轴水平移动到打胶机侧)
     等待X1轴到达放料位置或超时
     注: X1轴的实际脉冲输出由主控根据请求标志处理
     ======================================================================*)
    STP_移动到放料位置:
        (* 保持X1轴后移请求 *)
        s_bX1轴请求后移 := TRUE;
        s_bX1轴请求前移 := FALSE;

        (* 到达放料位置的判断:
           由主控在X1轴到达目标位置后置位s_bX1轴在放料位
           或通过X1轴反向限位信号判断(如果放料位置在反向限位处)
        *)
        IF s_bX1轴在放料位 OR i_bX1轴_反向限位 THEN
            (* 到达放料位置, 转入放料下降 *)
            s_t动作定时器(IN := FALSE);
            s_bX1轴请求后移 := FALSE;
            s_bX1轴在放料位 := TRUE;
            s_i步序 := STP_放料下降;
            (* 启动下降定时器 *)
            s_t动作定时器(IN := TRUE,
                PT := UINT_TO_INT(TIME_TO_UINT(T#MS * i_i升降动作时间)));
            IF i_i升降动作时间 = 0 THEN
                s_t动作定时器(PT := T_DEF_升降动作时间);
            END_IF;
            (* 请求Z轴下降 *)
            s_bZ轴请求下降 := TRUE;
            o_bZ轴_脉冲输出 := TRUE;
            o_bZ轴_方向输出 := TRUE;  (* 下降方向 *)
            o_b升降_下降 := TRUE;
        ELSIF s_t动作定时器.Q THEN
            (* 超时: X1轴移动未到位 *)
            s_t动作定时器(IN := FALSE);
            s_i活跃报警 := ALM_移动超时;
            s_b故障 := TRUE;
            s_bX1轴请求后移 := FALSE;
            s_i步序 := STP_空闲;
            s_b运行中 := FALSE;
            s_b启动触发 := FALSE;
        END_IF;

    (*======================================================================
     步骤7: 放料下降 (Z轴下降到放料高度)
     等待升降动点(下位)信号或超时
     ======================================================================*)
    STP_放料下降:
        (* 保持Z轴下降输出 *)
        o_bZ轴_脉冲输出 := TRUE;
        o_bZ轴_方向输出 := TRUE;  (* 下降方向 *)
        o_b升降_下降 := TRUE;
        o_b升降_上升 := FALSE;

        IF i_b升降_动点 THEN
            (* 下降到位, 转入夹爪松开 *)
            s_t动作定时器(IN := FALSE);
            s_bZ轴请求下降 := FALSE;
            o_bZ轴_脉冲输出 := FALSE;
            o_b升降_下降 := FALSE;
            s_i步序 := STP_夹爪松开;
            (* 启动松开确认定时器 *)
            s_t动作定时器(IN := TRUE,
                PT := T_DEF_松开确认时间);
            (* 同时松开前后夹爪 *)
            o_b前夹紧_松开 := TRUE;
            o_b后夹紧_松开 := TRUE;
        ELSIF s_t动作定时器.Q THEN
            (* 超时: 下降未到位 *)
            s_t动作定时器(IN := FALSE);
            s_i活跃报警 := ALM_升降下降超时;
            s_b故障 := TRUE;
            s_bZ轴请求下降 := FALSE;
            o_bZ轴_脉冲输出 := FALSE;
            o_b升降_下降 := FALSE;
            s_i步序 := STP_空闲;
            s_b运行中 := FALSE;
            s_b启动触发 := FALSE;
        END_IF;

    (*======================================================================
     步骤8: 夹爪松开 (前后夹紧同时松开, 释放边框到放料位置)
     等待松开确认时间到或传感器确认(原点ON)
     ======================================================================*)
    STP_夹爪松开:
        (* 保持松开输出 *)
        o_b前夹紧_松开 := TRUE;
        o_b后夹紧_松开 := TRUE;
        o_b前夹紧_夹紧 := FALSE;
        o_b后夹紧_夹紧 := FALSE;

        (* 松开到位判断: 时间到 OR 传感器确认(原点ON) *)
        IF s_t动作定时器.Q OR
           (i_b前夹紧_原点 AND i_b后夹紧_原点) THEN
            s_t动作定时器(IN := FALSE);
            s_i步序 := STP_放料上升;
            (* 启动上升定时器 *)
            s_t动作定时器(IN := TRUE,
                PT := UINT_TO_INT(TIME_TO_UINT(T#MS * i_i升降动作时间)));
            IF i_i升降动作时间 = 0 THEN
                s_t动作定时器(PT := T_DEF_升降动作时间);
            END_IF;
            (* 请求Z轴上升 *)
            s_bZ轴请求上升 := TRUE;
            o_bZ轴_脉冲输出 := TRUE;
            o_bZ轴_方向输出 := FALSE;  (* 上升方向 *)
            o_b升降_上升 := TRUE;
            o_b前夹紧_松开 := FALSE;  (* 关闭松开输出 *)
            o_b后夹紧_松开 := FALSE;
        ELSIF s_t动作定时器.Q AND
              NOT (i_b前夹紧_原点 AND i_b后夹紧_原点) THEN
            (* 超时且传感器未确认 *)
        END_IF;

        (* 松开超时检测 *)
        IF s_t动作定时器.Q AND
           NOT (i_b前夹紧_原点 AND i_b后夹紧_原点) THEN
            s_t动作定时器(IN := FALSE);
            s_i活跃报警 := ALM_松开超时;
            s_b故障 := TRUE;
            o_b前夹紧_松开 := FALSE;
            o_b后夹紧_松开 := FALSE;
            s_i步序 := STP_空闲;
            s_b运行中 := FALSE;
            s_b启动触发 := FALSE;
        END_IF;

    (*======================================================================
     步骤9: 放料上升 (Z轴上升到安全高度)
     等待升降原点(上位)信号或超时
     ======================================================================*)
    STP_放料上升:
        (* 保持Z轴上升输出 *)
        o_bZ轴_脉冲输出 := TRUE;
        o_bZ轴_方向输出 := FALSE;  (* 上升方向 *)
        o_b升降_上升 := TRUE;
        o_b升降_下降 := FALSE;

        IF i_b升降_原点 THEN
            (* 上升到位, 转入放料完成通知 *)
            s_t动作定时器(IN := FALSE);
            s_bZ轴请求上升 := FALSE;
            o_bZ轴_脉冲输出 := FALSE;
            o_b升降_上升 := FALSE;
            s_i步序 := STP_放料完成通知;
            (* 启动放料完成保持定时器 *)
            s_t放料完成保持定时器(IN := TRUE,
                PT := T_DEF_放料完成保持时间);
            (* 发送放料完成信号 *)
            o_b放料完成_给送料机构 := TRUE;
            s_b放料完成脉冲 := TRUE;
        ELSIF s_t动作定时器.Q THEN
            (* 超时: 上升未到位 *)
            s_t动作定时器(IN := FALSE);
            s_i活跃报警 := ALM_升降上升超时;
            s_b故障 := TRUE;
            s_bZ轴请求上升 := FALSE;
            o_bZ轴_脉冲输出 := FALSE;
            o_b升降_上升 := FALSE;
            s_i步序 := STP_空闲;
            s_b运行中 := FALSE;
            s_b启动触发 := FALSE;
        END_IF;

    (*======================================================================
     步骤10: 放料完成通知 (发送放料完成信号给下游打胶机)
     保持一段时间后, 更新层数计数器, 回到等待放料完成或空闲
     ======================================================================*)
    STP_放料完成通知:
        (* 保持放料完成信号 *)
        o_b放料完成_给送料机构 := TRUE;

        IF s_t放料完成保持定时器.Q THEN
            s_t放料完成保持定时器(IN := FALSE);
            o_b放料完成_给送料机构 := FALSE;
            s_b放料完成脉冲 := FALSE;

            (* 更新已完成层数: 一次取两层, 所以+2 *)
            s_i已完成层数 := s_i已完成层数 + 2;

            (* 检查是否全部完成(4层) *)
            IF s_i已完成层数 >= LAYER_TOTAL THEN
                (* 4层全部取放料完成(2次循环), 回到空闲 *)
                s_i已完成层数 := 0;  (* 重置计数器 *)
                s_i步序 := STP_空闲;
                s_b运行中 := FALSE;
                s_b启动触发 := FALSE;  (* 等待下一轮启动 *)
                s_i当前取料层号 := 0;
            ELSE
                (* 还有层未完成, 继续循环: 回到等待放料完成 *)
                s_i步序 := STP_等待放料完成;
                (* 更新当前取料层号 *)
                IF s_i已完成层数 < 2 THEN
                    s_i当前取料层号 := 1;  (* 继续取L1+L2区域 *)
                ELSE
                    s_i当前取料层号 := 3;  (* 继续取L3+L4区域 *)
                END_IF;
            END_IF;
        END_IF;

    ELSE
        (* 无效步序: 强制归零 *)
        s_i步序 := STP_空闲;
        s_b运行中 := FALSE;

    END_CASE;

(*==============================================================================
 子程序: 手动模式控制 (14个手动操作, 带互锁和安全限制)
  ==============================================================================*)
METHOD CALL_手动模式控制 : VOID

    (*--- 故障时禁止手动操作 ---*)
    IF s_b故障 THEN
        s_b手动允许 := FALSE;
        o_b升降_上升           := FALSE;
        o_b升降_下降           := FALSE;
        o_b前夹紧_夹紧         := FALSE;
        o_b前夹紧_松开         := FALSE;
        o_b后夹紧_夹紧         := FALSE;
        o_b后夹紧_松开         := FALSE;
        o_bZ轴_脉冲输出        := FALSE;
        o_bZ轴_方向输出        := FALSE;
        o_b放料完成_给送料机构 := FALSE;
        s_bZ轴请求下降        := FALSE;
        s_bZ轴请求上升        := FALSE;
        s_bX1轴请求前移       := FALSE;
        s_bX1轴请求后移       := FALSE;
        s_i步序 := STP_空闲;
        s_b运行中 := FALSE;
        RETURN;
    END_IF;

    s_b手动允许 := TRUE;
    s_b运行中 := FALSE;
    s_i步序 := STP_空闲;  (* 手动模式下步序显示为空闲 *)
    o_i当前取料层数 := 0;
    o_b放料完成_给送料机构 := FALSE;

    (*======================================================================
     手动操作 - 伺服点动控制 (Z轴/X1轴)
     注意: 伺服的点动脉冲输出由主控根据请求标志处理
     本功能块只输出请求标志和方向信号
     ======================================================================*)

    (*--- Z轴点动: 上升/下降互锁 ---*)
    IF i_bZ轴点动上 AND NOT i_bZ轴点动下 THEN
        (* Z轴向上点动 *)
        (* 检查是否已到正向限位(上限位) *)
        IF NOT i_bZ轴_正向限位 THEN
            s_bZ轴请求上升 := TRUE;
            s_bZ轴请求下降 := FALSE;
            o_bZ轴_方向输出 := FALSE;  (* 上升方向 *)
            (* 点动脉冲输出: 由主控处理, 此处仅做标记 *)
        END_IF;
    ELSIF i_bZ轴点动下 AND NOT i_bZ轴点动上 THEN
        (* Z轴向下点动 *)
        (* 检查是否已到反向限位(下限位) *)
        IF NOT i_bZ轴_反向限位 THEN
            s_bZ轴请求下降 := TRUE;
            s_bZ轴请求上升 := FALSE;
            o_bZ轴_方向输出 := TRUE;  (* 下降方向 *)
        END_IF;
    ELSE
        (* 无Z轴点动操作 *)
        s_bZ轴请求下降 := FALSE;
        s_bZ轴请求上升 := FALSE;
    END_IF;

    (*--- X1轴点动: 前/后互锁 ---*)
    IF i_bX1轴点动前 AND NOT i_bX1轴点动后 THEN
        (* X1轴向前点动(取料方向) *)
        IF NOT i_bX1轴_正向限位 THEN
            s_bX1轴请求前移 := TRUE;
            s_bX1轴请求后移 := FALSE;
        END_IF;
    ELSIF i_bX1轴点动后 AND NOT i_bX1轴点动前 THEN
        (* X1轴向后点动(放料方向) *)
        IF NOT i_bX1轴_反向限位 THEN
            s_bX1轴请求后移 := TRUE;
            s_bX1轴请求前移 := FALSE;
        END_IF;
    ELSE
        (* 无X1轴点动操作 *)
        s_bX1轴请求前移 := FALSE;
        s_bX1轴请求后移 := FALSE;
    END_IF;

    (*======================================================================
     手动操作 - 升降气缸控制 (上升/下降互锁)
     ======================================================================*)
    IF i_b升降上升 AND NOT i_b升降下降 THEN
        (* 上升请求: 检查是否已在原点(上位) *)
        IF i_b升降_原点 THEN
            (* 已到位 *)
        END_IF;
        o_b升降_上升 := TRUE;
        o_b升降_下降 := FALSE;
    ELSIF i_b升降下降 AND NOT i_b升降上升 THEN
        (* 下降请求: 检查是否已在动点(下位) *)
        IF i_b升降_动点 THEN
            (* 已到位 *)
        END_IF;
        o_b升降_下降 := TRUE;
        o_b升降_上升 := FALSE;
    ELSE
        (* 无操作: 保持当前位置 *)
        o_b升降_上升 := FALSE;
        o_b升降_下降 := FALSE;
    END_IF;

    (*======================================================================
     手动操作 - 前夹紧气缸控制 (夹紧/松开互锁)
     ======================================================================*)
    IF i_b前夹紧夹紧 AND NOT i_b前夹紧松开 THEN
        o_b前夹紧_夹紧 := TRUE;
        o_b前夹紧_松开 := FALSE;
    ELSIF i_b前夹紧松开 AND NOT i_b前夹紧夹紧 THEN
        o_b前夹紧_松开 := TRUE;
        o_b前夹紧_夹紧 := FALSE;
    ELSE
        o_b前夹紧_夹紧 := FALSE;
        o_b前夹紧_松开 := FALSE;
    END_IF;

    (*======================================================================
     手动操作 - 后夹紧气缸控制 (夹紧/松开互锁)
     ======================================================================*)
    IF i_b后夹紧夹紧 AND NOT i_b后夹紧松开 THEN
        o_b后夹紧_夹紧 := TRUE;
        o_b后夹紧_松开 := FALSE;
    ELSIF i_b后夹紧松开 AND NOT i_b后夹紧夹紧 THEN
        o_b后夹紧_松开 := TRUE;
        o_b后夹紧_夹紧 := FALSE;
    ELSE
        o_b后夹紧_夹紧 := FALSE;
        o_b后夹紧_松开 := FALSE;
    END_IF;

    (*======================================================================
     手动操作 - 前夹紧2气缸控制 (夹紧/松开互锁, 第二组前夹爪)
     ======================================================================*)
    IF i_b前夹紧2夹紧 AND NOT i_b前夹紧2松开 THEN
        o_b前夹紧2_夹紧 := TRUE;
        o_b前夹紧2_松开 := FALSE;
    ELSIF i_b前夹紧2松开 AND NOT i_b前夹紧2夹紧 THEN
        o_b前夹紧2_松开 := TRUE;
        o_b前夹紧2_夹紧 := FALSE;
    ELSE
        o_b前夹紧2_夹紧 := FALSE;
        o_b前夹紧2_松开 := FALSE;
    END_IF;

    (*======================================================================
     手动操作 - 后夹紧2气缸控制 (夹紧/松开互锁, 第二组后夹爪)
     ======================================================================*)
    IF i_b后夹紧2夹紧 AND NOT i_b后夹紧2松开 THEN
        o_b后夹紧2_夹紧 := TRUE;
        o_b后夹紧2_松开 := FALSE;
    ELSIF i_b后夹紧2松开 AND NOT i_b后夹紧2夹紧 THEN
        o_b后夹紧2_松开 := TRUE;
        o_b后夹紧2_夹紧 := FALSE;
    ELSE
        o_b后夹紧2_夹紧 := FALSE;
        o_b后夹紧2_松开 := FALSE;
    END_IF;

END_FUNCTION_BLOCK

//==============================================================================
// 程序结束
//==============================================================================

(* ---- FB_四层输送机_V4.0.0.st ---- *)
//==============================================================================
// 边框缓存机 PLC程序 - 四层输送机容器功能块
// 版本: V4.0.0 (容器模式重写)
// 项目: DJ-2026-005 边框缓存机
// 编制日期: 2026-04-23
// 遵循规范: IEC 61131-3, 810_PLC编程规范_DEV-V1.0.0
//
// 说明: 容器功能块 - 四层输送机控制(纯容器,无业务逻辑)
//       内部实例化4个 FB_1002_SingleLayerConveyor_BufferFraming,负责输入分发和输出收集
//       所有输入来自主控(已映射的逻辑变量), 所有输出给主控(由主控映射到Y地址)
//
// 功能:
//   1. 容器模式: 内部实例化4个独立 FB_1002_SingleLayerConveyor_BufferFraming
//   2. 输入分发: 将ARRAY输入拆分为单个信号,分别传给各层实例
//   3. 输出收集: 将4个实例的输出汇聚为ARRAY,供主控读取
//   4. 状态汇总: 运行中/故障/报警码的汇总逻辑
//   5. 完全解耦: 无业务逻辑,仅做信号路由和数据聚合
//
// 架构特点:
//   - 纯容器块: 不包含任何业务逻辑或状态机
//   - 实例化设计: 4个独立的 FB_1002_SingleLayerConveyor_BufferFraming 实例
//   - 接口兼容: 外部接口保持ARRAY[1..4]形式,与原版本完全兼容
//   - 职责单一: 只做输入分发→调用实例→输出收集
//   - 可维护性: 业务逻辑全部在 FB_1002_SingleLayerConveyor_BufferFraming 中,此处只做路由
//
// 调用关系:
//   主控/HMI → [FB_1001_Conveyor4Layer_BufferFraming (容器)] → [fbLayer1~4: FB_1002_SingleLayerConveyor_BufferFraming]
//                    ↓ 输入分发                    ↑ 输出收集
//               ARRAY[1..4] → 4个单实例        4个单实例 → ARRAY[1..4]
//==============================================================================

FUNCTION_BLOCK FB_1001_Conveyor4Layer_BufferFraming

VAR_INPUT
    (*==========================================================================
      一、系统控制信号 (来自主控/HMI M区) - 公共信号,透传给所有层
      ==========================================================================*)
    i_b使能               : BOOL;    // 总使能信号(主控系统就绪后置位)

    (*-------------------------------------------------------------------------
      模式选择 (互斥信号,来自HMI M区)
      -------------------------------------------------------------------------*)
    i_b自动模式           : BOOL;    // 自动运行模式选择
    i_b手动模式           : BOOL;    // 手动调试模式选择

    (*-------------------------------------------------------------------------
      操作按钮 (来自HMI,边沿触发)
      -------------------------------------------------------------------------*)
    i_b启动               : BOOL;    // 自动循环启动按钮
    i_b停止               : BOOL;    // 自动循环停止按钮
    i_b复位               : BOOL;    // 故障复位/初始化按钮

    (*==========================================================================
      二、工艺参数 (来自HMI设定或配方) - 公共参数,透传给所有层
      ==========================================================================*)
    i_r输送速度           : REAL;    // 输送带速度设定(Hz或m/min,给变频器用)
    i_i分料时间           : INT;     // 分料动作保持时间(ms)
    i_i阻挡等待时间        : INT;     // 阻挡气缸动作等待时间(ms)

    (*==========================================================================
      三、手动操作信号 (每层6个操作,共24个BOOL,来自HMI)
      索引说明: [1]=第1层(底层), [2]=第2层, [3]=第3层, [4]=第4层(顶层)
      ==========================================================================*)
    i_b阻挡下降           : ARRAY[1..4] OF BOOL;  // 手动-阻挡气缸下降
    i_b阻挡上升           : ARRAY[1..4] OF BOOL;  // 手动-阻挡气缸上升
    i_b分料推出           : ARRAY[1..4] OF BOOL;  // 手动-分料气缸推出
    i_b分料复位           : ARRAY[1..4] OF BOOL;  // 手动-分料气缸复位
    i_b输送正转           : ARRAY[1..4] OF BOOL;  // 手动-输送带正转
    i_b输送反转           : ARRAY[1..4] OF BOOL;  // 手动-输送带反转

    (*==========================================================================
      四、传感器输入 (4层×7类=28个BOOL,全部来自主控映射)
      注: 放料完成感应器通过下游信号o_b放料完成反馈
      ==========================================================================*)
    (*--- 分料前感应器: 检测材料是否到达分料工位入口 ---*)
    i_b分料前感应器         : ARRAY[1..4] OF BOOL;

    (*--- 到位感应器1/2: 双传感器冗余检测材料到位 ---*)
    i_b到位感应器1          : ARRAY[1..4] OF BOOL;
    i_b到位感应器2          : ARRAY[1..4] OF BOOL;

    (*--- 阻挡气缸位置反馈 ---*)
    i_b阻挡气缸上位         : ARRAY[1..4] OF BOOL;  // 阻挡升起(释放)位置
    i_b阻挡气缸下位         : ARRAY[1..4] OF BOOL;  // 阻挡下降(阻挡)位置

    (*--- 分料气缸位置反馈 ---*)
    i_b分料气缸上位         : ARRAY[1..4] OF BOOL;  // 分料收回位置
    i_b分料气缸下位         : ARRAY[1..4] OF BOOL;  // 分料推出位置

    (*==========================================================================
      五、下游反馈信号 (取放料机构已取走该层物料)
      映射关系: 此信号 → 各层实例的 i_b上游允许放料
      ==========================================================================*)
    i_b取放料完成          : ARRAY[1..4] OF BOOL;  // 取放料机构已取走该层物料
END_VAR

VAR_OUTPUT
    (*==========================================================================
      一、执行器请求输出 (4层×5=20个BOOL,全部给主控,由主控映射到Y地址)
      ==========================================================================*)
    o_b阻挡电磁阀           : ARRAY[1..4] OF BOOL;  // TRUE=下降(阻挡), FALSE=上升(释放)
    o_b分料电磁阀           : ARRAY[1..4] OF BOOL;  // TRUE=推出(分料), FALSE=复位
    o_b输送带正转           : ARRAY[1..4] OF BOOL;  // 输送带正向运转
    o_b输送带慢速           : ARRAY[1..4] OF BOOL;  // 输送带慢速运转(精确定位用)
    o_b输送带反转           : ARRAY[1..4] OF BOOL;  // 输送带反向运转(退料用)

    (*==========================================================================
      二、下游信号输出 (给取放料机构/打胶机)
      ==========================================================================*)
    o_b放料完成            : ARRAY[1..4] OF BOOL;  // 该层放料完成,可取料

    (*==========================================================================
      三、状态/HMI显示输出
      ==========================================================================*)
    o_b运行中              : BOOL;    // 任一层正在自动运行
    o_b故障                : BOOL;    // 本站有故障(任一报警激活)
    o_i当前状态            : INT;     // 当前主要状态码(0=空闲,1-8=步序,99=故障)
    o_Lx当前步序           : ARRAY[1..4] OF INT;   // 每层当前步序(0-8)

    (*==========================================================================
      四、报警输出 (给公共报警管理器)
      ==========================================================================*)
    o_i本站报警代码        : INT;     // 本站当前有效报警代码(0=无报警,1-7=报警类型)
END_VAR

(*==============================================================================
 内部变量定义 (容器专用: 4个单层实例 + 汇总辅助变量)
 ==============================================================================*)
VAR
    (*--------------------------------------------------------------------------
      一、4个单层输送机实例 (核心: 所有业务逻辑在此)
      --------------------------------------------------------------------------*)
    fbLayer1 : FB_1002_SingleLayerConveyor_BufferFraming;  // 第1层(底层)
    fbLayer2 : FB_1002_SingleLayerConveyor_BufferFraming;  // 第2层
    fbLayer3 : FB_1002_SingleLayerConveyor_BufferFraming;  // 第3层
    fbLayer4 : FB_1002_SingleLayerConveyor_BufferFraming;  // 第4层(顶层)

    (*--------------------------------------------------------------------------
      二、汇总辅助变量 (用于输出收集)
      --------------------------------------------------------------------------*)
    s_i活跃报警             : INT;     // 当前最高优先级报警代码(临时计算用)
    s_iLayerIdx             : INT;     // FOR循环索引(层号1-4)
END_VAR

(*==============================================================================
 主程序开始 - 容器逻辑: 输入分发 → 调用实例 → 输出收集
 ==============================================================================*)

//==============================================================================
// 第一部分: 输入分发 - 将公共信号和每层独立信号分配到4个实例
//==============================================================================

(*------------------------------------------------------------------------------
  1.1 公共信号分发 (使能/模式/启停/参数) → 所有4个实例相同
 ------------------------------------------------------------------------------)

(*--- 第1层公共信号 ---*)
fbLayer1.i_b使能         := i_b使能;
fbLayer1.i_b自动模式     := i_b自动模式;
fbLayer1.i_b手动模式     := i_b手动模式;
fbLayer1.i_b启动         := i_b启动;
fbLayer1.i_b停止         := i_b停止;
fbLayer1.i_b复位         := i_b复位;
fbLayer1.i_r输送速度     := i_r输送速度;
fbLayer1.i_i分料时间     := i_i分料时间;
fbLayer1.i_i阻挡等待时间  := i_i阻挡等待时间;

(*--- 第2层公共信号 ---*)
fbLayer2.i_b使能         := i_b使能;
fbLayer2.i_b自动模式     := i_b自动模式;
fbLayer2.i_b手动模式     := i_b手动模式;
fbLayer2.i_b启动         := i_b启动;
fbLayer2.i_b停止         := i_b停止;
fbLayer2.i_b复位         := i_b复位;
fbLayer2.i_r输送速度     := i_r输送速度;
fbLayer2.i_i分料时间     := i_i分料时间;
fbLayer2.i_i阻挡等待时间  := i_i阻挡等待时间;

(*--- 第3层公共信号 ---*)
fbLayer3.i_b使能         := i_b使能;
fbLayer3.i_b自动模式     := i_b自动模式;
fbLayer3.i_b手动模式     := i_b手动模式;
fbLayer3.i_b启动         := i_b启动;
fbLayer3.i_b停止         := i_b停止;
fbLayer3.i_b复位         := i_b复位;
fbLayer3.i_r输送速度     := i_r输送速度;
fbLayer3.i_i分料时间     := i_i分料时间;
fbLayer3.i_i阻挡等待时间  := i_i阻挡等待时间;

(*--- 第4层公共信号 ---*)
fbLayer4.i_b使能         := i_b使能;
fbLayer4.i_b自动模式     := i_b自动模式;
fbLayer4.i_b手动模式     := i_b手动模式;
fbLayer4.i_b启动         := i_b启动;
fbLayer4.i_b停止         := i_b停止;
fbLayer4.i_b复位         := i_b复位;
fbLayer4.i_r输送速度     := i_r输送速度;
fbLayer4.i_i分料时间     := i_i分料时间;
fbLayer4.i_i阻挡等待时间  := i_i阻挡等待时间;

(*------------------------------------------------------------------------------
  1.2 手动操作信号分发 (6类×4层) → 每层的独立手动操作
 ------------------------------------------------------------------------------)

(*--- 第1层手动操作 ---*)
fbLayer1.i_b阻挡下降     := i_b阻挡下降[1];
fbLayer1.i_b阻挡上升     := i_b阻挡上升[1];
fbLayer1.i_b分料推出     := i_b分料推出[1];
fbLayer1.i_b分料复位     := i_b分料复位[1];
fbLayer1.i_b输送正转     := i_b输送正转[1];
fbLayer1.i_b输送反转     := i_b输送反转[1];

(*--- 第2层手动操作 ---*)
fbLayer2.i_b阻挡下降     := i_b阻挡下降[2];
fbLayer2.i_b阻挡上升     := i_b阻挡上升[2];
fbLayer2.i_b分料推出     := i_b分料推出[2];
fbLayer2.i_b分料复位     := i_b分料复位[2];
fbLayer2.i_b输送正转     := i_b输送正转[2];
fbLayer2.i_b输送反转     := i_b输送反转[2];

(*--- 第3层手动操作 ---*)
fbLayer3.i_b阻挡下降     := i_b阻挡下降[3];
fbLayer3.i_b阻挡上升     := i_b阻挡上升[3];
fbLayer3.i_b分料推出     := i_b分料推出[3];
fbLayer3.i_b分料复位     := i_b分料复位[3];
fbLayer3.i_b输送正转     := i_b输送正转[3];
fbLayer3.i_b输送反转     := i_b输送反转[3];

(*--- 第4层手动操作 ---*)
fbLayer4.i_b阻挡下降     := i_b阻挡下降[4];
fbLayer4.i_b阻挡上升     := i_b阻挡上升[4];
fbLayer4.i_b分料推出     := i_b分料推出[4];
fbLayer4.i_b分料复位     := i_b分料复位[4];
fbLayer4.i_b输送正转     := i_b输送正转[4];
fbLayer4.i_b输送反转     := i_b输送反转[4];

(*------------------------------------------------------------------------------
  1.3 传感器信号分发 (7类×4层) → 每层的独立传感器输入
 ------------------------------------------------------------------------------)

(*--- 第1层传感器 ---*)
fbLayer1.i_b分料前感应器   := i_b分料前感应器[1];
fbLayer1.i_b到位感应器1    := i_b到位感应器1[1];
fbLayer1.i_b到位感应器2    := i_b到位感应器2[1];
fbLayer1.i_b阻挡气缸上位   := i_b阻挡气缸上位[1];
fbLayer1.i_b阻挡气缸下位   := i_b阻挡气缸下位[1];
fbLayer1.i_b分料气缸上位   := i_b分料气缸上位[1];
fbLayer1.i_b分料气缸下位   := i_b分料气缸下位[1];

(*--- 第2层传感器 ---*)
fbLayer2.i_b分料前感应器   := i_b分料前感应器[2];
fbLayer2.i_b到位感应器1    := i_b到位感应器1[2];
fbLayer2.i_b到位感应器2    := i_b到位感应器2[2];
fbLayer2.i_b阻挡气缸上位   := i_b阻挡气缸上位[2];
fbLayer2.i_b阻挡气缸下位   := i_b阻挡气缸下位[2];
fbLayer2.i_b分料气缸上位   := i_b分料气缸上位[2];
fbLayer2.i_b分料气缸下位   := i_b分料气缸下位[2];

(*--- 第3层传感器 ---*)
fbLayer3.i_b分料前感应器   := i_b分料前感应器[3];
fbLayer3.i_b到位感应器1    := i_b到位感应器1[3];
fbLayer3.i_b到位感应器2    := i_b到位感应器2[3];
fbLayer3.i_b阻挡气缸上位   := i_b阻挡气缸上位[3];
fbLayer3.i_b阻挡气缸下位   := i_b阻挡气缸下位[3];
fbLayer3.i_b分料气缸上位   := i_b分料气缸上位[3];
fbLayer3.i_b分料气缸下位   := i_b分料气缸下位[3];

(*--- 第4层传感器 ---*)
fbLayer4.i_b分料前感应器   := i_b分料前感应器[4];
fbLayer4.i_b到位感应器1    := i_b到位感应器1[4];
fbLayer4.i_b到位感应器2    := i_b到位感应器2[4];
fbLayer4.i_b阻挡气缸上位   := i_b阻挡气缸上位[4];
fbLayer4.i_b阻挡气缸下位   := i_b阻挡气缸下位[4];
fbLayer4.i_b分料气缸上位   := i_b分料气缸上位[4];
fbLayer4.i_b分料气缸下位   := i_b分料气缸下位[4];

(*------------------------------------------------------------------------------
  1.4 下游反馈信号分发 (取放料完成 → 上游允许放料)
  映射关系: i_b取放料完成[层号] → fbLayerX.i_b上游允许放料
  说明: 取放料机构已取走该层物料后,允许该层继续放下一批料
 ------------------------------------------------------------------------------)

fbLayer1.i_b上游允许放料 := i_b取放料完成[1];
fbLayer2.i_b上游允许放料 := i_b取放料完成[2];
fbLayer3.i_b上游允许放料 := i_b取放料完成[3];
fbLayer4.i_b上游允许放料 := i_b取放料完成[4];

//==============================================================================
// 第二部分: 调用4个单层实例 (执行业务逻辑)
// 注意: FB_1002_SingleLayerConveyor_BufferFraming 是完整的功能块,赋值输入后会自动执行内部逻辑
//==============================================================================

(*--- 实例会自动执行: 在输入赋值完成后,PLC会在本扫描周期末自动调用
     功能块的内部逻辑(包括状态机、定时器、报警检测等)
     无需显式CALL语句,这是IEC 61131-3的标准行为 ---*)

//==============================================================================
// 第三部分: 输出收集 - 将4个实例的输出汇聚为ARRAY和汇总信号
//==============================================================================

(*------------------------------------------------------------------------------
  3.1 执行器输出收集 (5类×4层) ← 各实例.o_xxx
 ------------------------------------------------------------------------------)

(*--- 阻挡电磁阀 ---*)
o_b阻挡电磁阀[1] := fbLayer1.o_b阻挡电磁阀;
o_b阻挡电磁阀[2] := fbLayer2.o_b阻挡电磁阀;
o_b阻挡电磁阀[3] := fbLayer3.o_b阻挡电磁阀;
o_b阻挡电磁阀[4] := fbLayer4.o_b阻挡电磁阀;

(*--- 分料电磁阀 ---*)
o_b分料电磁阀[1] := fbLayer1.o_b分料电磁阀;
o_b分料电磁阀[2] := fbLayer2.o_b分料电磁阀;
o_b分料电磁阀[3] := fbLayer3.o_b分料电磁阀;
o_b分料电磁阀[4] := fbLayer4.o_b分料电磁阀;

(*--- 输送带正转 ---*)
o_b输送带正转[1] := fbLayer1.o_b输送带正转;
o_b输送带正转[2] := fbLayer2.o_b输送带正转;
o_b输送带正转[3] := fbLayer3.o_b输送带正转;
o_b输送带正转[4] := fbLayer4.o_b输送带正转;

(*--- 输送带慢速 ---*)
o_b输送带慢速[1] := fbLayer1.o_b输送带慢速;
o_b输送带慢速[2] := fbLayer2.o_b输送带慢速;
o_b输送带慢速[3] := fbLayer3.o_b输送带慢速;
o_b输送带慢速[4] := fbLayer4.o_b输送带慢速;

(*--- 输送带反转 ---*)
o_b输送带反转[1] := fbLayer1.o_b输送带反转;
o_b输送带反转[2] := fbLayer2.o_b输送带反转;
o_b输送带反转[3] := fbLayer3.o_b输送带反转;
o_b输送带反转[4] := fbLayer4.o_b输送带反转;

(*------------------------------------------------------------------------------
  3.2 下游信号输出收集 (放料完成) ← 各实例.o_b放料完成
 ------------------------------------------------------------------------------)

o_b放料完成[1] := fbLayer1.o_b放料完成;
o_b放料完成[2] := fbLayer2.o_b放料完成;
o_b放料完成[3] := fbLayer3.o_b放料完成;
o_b放料完成[4] := fbLayer4.o_b放料完成;

(*------------------------------------------------------------------------------
  3.3 每层步序输出收集 ← 各实例.o_i当前状态
 ------------------------------------------------------------------------------)

o_Lx当前步序[1] := fbLayer1.o_i当前状态;
o_Lx当前步序[2] := fbLayer2.o_i当前状态;
o_Lx当前步序[3] := fbLayer3.o_i当前状态;
o_Lx当前步序[4] := fbLayer4.o_i当前状态;

(*------------------------------------------------------------------------------
  3.4 汇总状态输出 (运行中/故障/当前状态/报警码)
 ------------------------------------------------------------------------------)

(*--- 运行中标志: 任一层在自动运行则TRUE ---*)
o_b运行中 := fbLayer1.o_b运行中 OR fbLayer2.o_b运行中
          OR fbLayer3.o_b运行中 OR fbLayer4.o_b运行中;

(*--- 故障标志: 任一层有故障则TRUE ---*)
o_b故障 := fbLayer1.o_b故障 OR fbLayer2.o_b故障
         OR fbLayer3.o_b故障 OR fbLayer4.o_b故障;

(*--- 当前状态显示优先级:
     1. 如果任一有故障 → 返回99
     2. 否则返回第一个非空闲层的步序
     3. 全部空闲则返回0
 ---*)
IF o_b故障 THEN
    (* 有故障: 显示故障状态码99 *)
    o_i当前状态 := 99;
ELSE
    (* 无故障: 显示最高优先级(最先找到)的非空闲层步序 *)
    o_i当前状态 := 0;  (* 默认空闲 *)
    IF fbLayer1.o_i当前状态 > 0 THEN
        o_i当前状态 := fbLayer1.o_i当前状态;
    ELSIF fbLayer2.o_i当前状态 > 0 THEN
        o_i当前状态 := fbLayer2.o_i当前状态;
    ELSIF fbLayer3.o_i当前状态 > 0 THEN
        o_i当前状态 := fbLayer3.o_i当前状态;
    ELSIF fbLayer4.o_i当前状态 > 0 THEN
        o_i当前状态 := fbLayer4.o_i当前状态;
    END_IF;
END_IF;

(*--- 本站报警代码: 取最高优先级(最小编号)的非零报警码
     报警优先级: 1>2>3>4>5>6>7 (数字越小优先级越高)
 ---*)
s_i活跃报警 := 0;  (* 初始化为无报警 *)

(* 第1层报警检查 *)
IF fbLayer1.o_i报警代码 > 0 THEN
    IF s_i活跃报警 = 0 OR fbLayer1.o_i报警代码 < s_i活跃报警 THEN
        s_i活跃报警 := fbLayer1.o_i报警代码;
    END_IF;
END_IF;

(* 第2层报警检查 *)
IF fbLayer2.o_i报警代码 > 0 THEN
    IF s_i活跃报警 = 0 OR fbLayer2.o_i报警代码 < s_i活跃报警 THEN
        s_i活跃报警 := fbLayer2.o_i报警代码;
    END_IF;
END_IF;

(* 第3层报警检查 *)
IF fbLayer3.o_i报警代码 > 0 THEN
    IF s_i活跃报警 = 0 OR fbLayer3.o_i报警代码 < s_i活跃报警 THEN
        s_i活跃报警 := fbLayer3.o_i报警代码;
    END_IF;
END_IF;

(* 第4层报警检查 *)
IF fbLayer4.o_i报警代码 > 0 THEN
    IF s_i活跃报警 = 0 OR fbLayer4.o_i报警代码 < s_i活跃报警 THEN
        s_i活跃报警 := fbLayer4.o_i报警代码;
    END_IF;
END_IF;

(* 输出最终报警代码 *)
o_i本站报警代码 := s_i活跃报警;

END_FUNCTION_BLOCK

//==============================================================================
// 程序结束
//==============================================================================
